LIN {X 0,Y 735.918,Z 1197.735,A -85,B 0,C 180,E1 27996.24,E2 27996.24} C_VEL
LIN {X 0,Y 735.912,Z 1201.928,A -85,B 0,C 180,E1 27994.051,E2 27994.051} C_VEL
LIN {X 0,Y 735.912,Z 1204.213,A -85,B 0,C 180,E1 27992.024,E2 27992.024} C_VEL
LIN {X 0,Y 735.898,Z 1204.939,A -85,B 0,C 180,E1 27989.766,E2 27989.766} C_VEL
LIN {X 0,Y 735.908,Z 1203.976,A -85,B 0,C 180,E1 27987.664,E2 27987.664} C_VEL
LIN {X 0,Y 735.91,Z 1201.303,A -85,B 0,C 180,E1 27985.558,E2 27985.558} C_VEL
LIN {X 0,Y 735.921,Z 1197.152,A -85,B 0,C 180,E1 27983.525,E2 27983.525} C_VEL
LIN {X 0,Y 735.931,Z 1191.15,A -85,B 0,C 180,E1 27981.405,E2 27981.405} C_VEL
LIN {X 0,Y 735.932,Z 1183.317,A -85,B 0,C 180,E1 27979.272,E2 27979.272} C_VEL
LIN {X 0,Y 735.999,Z 1173.523,A -85,B 0,C 180,E1 27977.126,E2 27977.126} C_VEL
LIN {X 0,Y 736.044,Z 1164.524,A -85,B 0,C 180,E1 27975.445,E2 27975.445} C_VEL
LIN {X 0,Y 736.091,Z 1154.647,A -85,B 0,C 180,E1 27973.817,E2 27973.817} C_VEL
LIN {X 0,Y 736.198,Z 1143.668,A -85,B 0,C 180,E1 27972.206,E2 27972.206} C_VEL
LIN {X 0,Y 736.364,Z 1129.285,A -85,B 0,C 180,E1 27970.321,E2 27970.321} C_VEL
LIN {X 0,Y 736.522,Z 1112.613,A -85,B 0,C 180,E1 27968.414,E2 27968.414} C_VEL
LIN {X 0,Y 736.685,Z 1097.971,A -85,B 0,C 180,E1 27966.905,E2 27966.905} C_VEL
LIN {X 0,Y 736.985,Z 1079.519,A -85,B 0,C 180,E1 27965.184,E2 27965.184} C_VEL
LIN {X 0,Y 737.229,Z 1060.157,A -85,B 0,C 180,E1 27963.586,E2 27963.586} C_VEL
LIN {X 0,Y 737.478,Z 1042.502,A -85,B 0,C 180,E1 27962.263,E2 27962.263} C_VEL
LIN {X 0,Y 737.894,Z 1020.414,A -85,B 0,C 180,E1 27960.77,E2 27960.77} C_VEL
LIN {X 0,Y 738.221,Z 997.825,A -85,B 0,C 180,E1 27959.43,E2 27959.43} C_VEL
LIN {X 0,Y 738.518,Z 977.714,A -85,B 0,C 180,E1 27958.361,E2 27958.361} C_VEL
LIN {X 0,Y 738.841,Z 956.603,A -85,B 0,C 180,E1 27957.36,E2 27957.36} C_VEL
LIN {X 0,Y 739.293,Z 929.665,A -85,B 0,C 180,E1 27956.257,E2 27956.257} C_VEL
LIN {X 0,Y 739.568,Z 907.021,A -85,B 0,C 180,E1 27955.471,E2 27955.471} C_VEL
LIN {X 0,Y 739.849,Z 883.645,A -85,B 0,C 180,E1 27954.779,E2 27954.779} C_VEL
LIN {X 0,Y 740.114,Z 856.949,A -85,B 0,C 180,E1 27954.147,E2 27954.147} C_VEL
LIN {X 0,Y 740.323,Z 829.837,A -85,B 0,C 180,E1 27953.669,E2 27953.669} C_VEL
LIN {X 0,Y 740.627,Z 742.145,A -85,B 0,C 180,E1 27952.618,E2 27952.618} C_VEL
LIN {X 0,Y 741.295,Z 519.857,A -85,B 0,C 180,E1 27949.955,E2 27949.955} C_VEL
LIN {X 0,Y 741.706,Z 355.878,A -85,B 0,C 180,E1 27947.919,E2 27947.919} C_VEL
LIN {X 0,Y 740.33,Z 349.95,A -85,B 0,C 180,E1 27947.733,E2 27947.733} C_VEL
LIN {X 0,Y 740.561,Z 322.858,A -85,B 0,C 180,E1 27946.081,E2 27946.081} C_VEL
LIN {X 0,Y 736.124,Z 312.939,A -85,B 0,C 180,E1 27945.097,E2 27945.097} C_VEL
LIN {X 0,Y 736.083,Z 312.459,A -85,B 0,C 180,E1 27944.721,E2 27944.721} C_VEL
LIN {X 0,Y 736.009,Z 312.546,A -85,B 0,C 180,E1 27941.944,E2 27941.944} C_VEL
LIN {X 0,Y 736.01,Z 312.538,A -85,B 0,C 180,E1 27939.58,E2 27939.58} C_VEL
LIN {X 0,Y 736.061,Z 312.541,A -85,B 0,C 180,E1 27936.989,E2 27936.989} C_VEL
LIN {X 0,Y 736.039,Z 312.539,A -85,B 0,C 180,E1 27934.035,E2 27934.035} C_VEL
LIN {X 0,Y 736.022,Z 312.539,A -85,B 0,C 180,E1 27931.536,E2 27931.536} C_VEL
LIN {X 0,Y 736.063,Z 312.544,A -85,B 0,C 180,E1 27928.921,E2 27928.921} C_VEL
LIN {X 0,Y 736.051,Z 312.538,A -85,B 0,C 180,E1 27925.853,E2 27925.853} C_VEL
LIN {X 0,Y 736.033,Z 312.534,A -85,B 0,C 180,E1 27923.286,E2 27923.286} C_VEL
LIN {X 0,Y 736.101,Z 312.542,A -85,B 0,C 180,E1 27920.515,E2 27920.515} C_VEL
LIN {X 0,Y 736.05,Z 312.53,A -85,B 0,C 180,E1 27917.552,E2 27917.552} C_VEL
LIN {X 0,Y 736.058,Z 312.542,A -85,B 0,C 180,E1 27914.877,E2 27914.877} C_VEL
LIN {X 0,Y 736.097,Z 312.528,A -85,B 0,C 180,E1 27911.916,E2 27911.916} C_VEL
LIN {X 0,Y 736.053,Z 312.538,A -85,B 0,C 180,E1 27909.145,E2 27909.145} C_VEL
LIN {X 0,Y 736.094,Z 312.534,A -85,B 0,C 180,E1 27906.317,E2 27906.317} C_VEL
LIN {X 0,Y 736.075,Z 312.534,A -85,B 0,C 180,E1 27903.349,E2 27903.349} C_VEL
LIN {X 0,Y 736.094,Z 312.536,A -85,B 0,C 180,E1 27900.389,E2 27900.389} C_VEL
LIN {X 0,Y 736.092,Z 312.531,A -85,B 0,C 180,E1 27897.353,E2 27897.353} C_VEL
LIN {X 0,Y 736.092,Z 312.536,A -85,B 0,C 180,E1 27894.309,E2 27894.309} C_VEL
LIN {X 0,Y 736.096,Z 312.53,A -85,B 0,C 180,E1 27891.249,E2 27891.249} C_VEL
LIN {X 0,Y 736.093,Z 312.53,A -85,B 0,C 180,E1 27889.116,E2 27889.116} C_VEL
LIN {X 0,Y 735.07,Z 312.665,A -85,B 0,C 180,E1 27888.516,E2 27888.516} C_VEL
LIN {X 0,Y 728.657,Z 313.451,A -85,B 0,C 180,E1 27886.837,E2 27886.837} C_VEL
LIN {X 0,Y 728.145,Z 313.52,A -85,B 0,C 180,E1 27886.401,E2 27886.401} C_VEL
LIN {X 0,Y 728.13,Z 313.524,A -85,B 0,C 180,E1 27883.567,E2 27883.567} C_VEL
LIN {X 0,Y 728.146,Z 313.517,A -85,B 0,C 180,E1 27880.674,E2 27880.674} C_VEL
LIN {X 0,Y 728.133,Z 313.526,A -85,B 0,C 180,E1 27877.75,E2 27877.75} C_VEL
LIN {X 0,Y 728.157,Z 313.518,A -85,B 0,C 180,E1 27874.806,E2 27874.806} C_VEL
LIN {X 0,Y 728.139,Z 313.522,A -85,B 0,C 180,E1 27871.811,E2 27871.811} C_VEL
LIN {X 0,Y 728.131,Z 313.525,A -85,B 0,C 180,E1 27868.913,E2 27868.913} C_VEL
LIN {X 0,Y 728.15,Z 313.526,A -85,B 0,C 180,E1 27865.831,E2 27865.831} C_VEL
LIN {X 0,Y 728.108,Z 313.521,A -85,B 0,C 180,E1 27863.023,E2 27863.023} C_VEL
LIN {X 0,Y 728.159,Z 313.531,A -85,B 0,C 180,E1 27860.139,E2 27860.139} C_VEL
LIN {X 0,Y 728.104,Z 313.534,A -85,B 0,C 180,E1 27857.281,E2 27857.281} C_VEL
LIN {X 0,Y 728.11,Z 313.537,A -85,B 0,C 180,E1 27854.655,E2 27854.655} C_VEL
LIN {X 0,Y 728.206,Z 313.843,A -85,B 0,C 180,E1 27853.987,E2 27853.987} C_VEL
LIN {X 0,Y 733.658,Z 326.305,A -85,B 0,C 180,E1 27852.727,E2 27852.727} C_VEL
LIN {X 0,Y 733.005,Z 366.435,A -85,B 0,C 180,E1 27850.182,E2 27850.182} C_VEL
LIN {X 0,Y 732.691,Z 396.674,A -85,B 0,C 180,E1 27848.329,E2 27848.329} C_VEL
LIN {X 0,Y 734.354,Z 404.868,A -85,B 0,C 180,E1 27848.118,E2 27848.118} C_VEL
LIN {X 0,Y 733.48,Z 650.838,A -85,B 0,C 180,E1 27845.227,E2 27845.227} C_VEL
LIN {X 0,Y 732.832,Z 829.718,A -85,B 0,C 180,E1 27843.161,E2 27843.161} C_VEL
LIN {X 0,Y 732.642,Z 853.04,A -85,B 0,C 180,E1 27842.782,E2 27842.782} C_VEL
LIN {X 0,Y 732.276,Z 879.242,A -85,B 0,C 180,E1 27842.196,E2 27842.196} C_VEL
LIN {X 0,Y 731.992,Z 900.709,A -85,B 0,C 180,E1 27841.591,E2 27841.591} C_VEL
LIN {X 0,Y 731.677,Z 923.398,A -85,B 0,C 180,E1 27840.828,E2 27840.828} C_VEL
LIN {X 0,Y 731.181,Z 948.746,A -85,B 0,C 180,E1 27839.807,E2 27839.807} C_VEL
LIN {X 0,Y 730.811,Z 969.465,A -85,B 0,C 180,E1 27838.835,E2 27838.835} C_VEL
LIN {X 0,Y 730.408,Z 992.417,A -85,B 0,C 180,E1 27837.606,E2 27837.606} C_VEL
LIN {X 0,Y 729.958,Z 1012.888,A -85,B 0,C 180,E1 27836.347,E2 27836.347} C_VEL
LIN {X 0,Y 729.623,Z 1031.699,A -85,B 0,C 180,E1 27835.053,E2 27835.053} C_VEL
LIN {X 0,Y 729.245,Z 1052.078,A -85,B 0,C 180,E1 27833.467,E2 27833.467} C_VEL
LIN {X 0,Y 728.963,Z 1068.5,A -85,B 0,C 180,E1 27832.033,E2 27832.033} C_VEL
LIN {X 0,Y 728.653,Z 1086.838,A -85,B 0,C 180,E1 27830.231,E2 27830.231} C_VEL
LIN {X 0,Y 728.464,Z 1101.019,A -85,B 0,C 180,E1 27828.652,E2 27828.652} C_VEL
LIN {X 0,Y 728.296,Z 1115.544,A -85,B 0,C 180,E1 27826.839,E2 27826.839} C_VEL
LIN {X 0,Y 728.144,Z 1127.947,A -85,B 0,C 180,E1 27825.042,E2 27825.042} C_VEL
LIN {X 0,Y 728.064,Z 1137.806,A -85,B 0,C 180,E1 27823.421,E2 27823.421} C_VEL
LIN {X 0,Y 728.005,Z 1147.195,A -85,B 0,C 180,E1 27821.648,E2 27821.648} C_VEL
LIN {X 0,Y 727.932,Z 1155.983,A -85,B 0,C 180,E1 27819.647,E2 27819.647} C_VEL
LIN {X 0,Y 727.933,Z 1162.049,A -85,B 0,C 180,E1 27817.957,E2 27817.957} C_VEL
LIN {X 0,Y 727.925,Z 1166.828,A -85,B 0,C 180,E1 27816.309,E2 27816.309} C_VEL
LIN {X 0,Y 727.903,Z 1171.167,A -85,B 0,C 180,E1 27814.333,E2 27814.333} C_VEL
LIN {X 0,Y 727.914,Z 1173.832,A -85,B 0,C 180,E1 27812.283,E2 27812.283} C_VEL
LIN {X 0,Y 727.892,Z 1174.814,A -85,B 0,C 180,E1 27810.63,E2 27810.63} C_VEL
LIN {X 0,Y 727.91,Z 1174.706,A -85,B 0,C 180,E1 27808.898,E2 27808.898} C_VEL
LIN {X 0,Y 727.905,Z 1172.917,A -85,B 0,C 180,E1 27806.772,E2 27806.772} C_VEL
LIN {X 0,Y 727.905,Z 1170.075,A -85,B 0,C 180,E1 27805.036,E2 27805.036} C_VEL
LIN {X 0,Y 727.912,Z 1166.237,A -85,B 0,C 180,E1 27803.374,E2 27803.374} C_VEL
LIN {X 0,Y 727.931,Z 1161.006,A -85,B 0,C 180,E1 27801.628,E2 27801.628} C_VEL
LIN {X 0,Y 727.963,Z 1152.715,A -85,B 0,C 180,E1 27799.474,E2 27799.474} C_VEL
LIN {X 0,Y 728.008,Z 1144.792,A -85,B 0,C 180,E1 27797.789,E2 27797.789} C_VEL
LIN {X 0,Y 728.062,Z 1135.921,A -85,B 0,C 180,E1 27796.161,E2 27796.161} C_VEL
LIN {X 0,Y 728.197,Z 1123.732,A -85,B 0,C 180,E1 27794.225,E2 27794.225} C_VEL
LIN {X 0,Y 728.327,Z 1111.132,A -85,B 0,C 180,E1 27792.503,E2 27792.503} C_VEL
LIN {X 0,Y 728.488,Z 1098.245,A -85,B 0,C 180,E1 27790.934,E2 27790.934} C_VEL
LIN {X 0,Y 728.768,Z 1081.226,A -85,B 0,C 180,E1 27789.101,E2 27789.101} C_VEL
LIN {X 0,Y 728.99,Z 1065.335,A -85,B 0,C 180,E1 27787.589,E2 27787.589} C_VEL
LIN {X 0,Y 729.358,Z 1046.931,A -85,B 0,C 180,E1 27786.017,E2 27786.017} C_VEL
LIN {X 0,Y 729.679,Z 1027.552,A -85,B 0,C 180,E1 27784.561,E2 27784.561} C_VEL
LIN {X 0,Y 730.105,Z 1007.614,A -85,B 0,C 180,E1 27783.22,E2 27783.22} C_VEL
LIN {X 0,Y 730.5,Z 985.362,A -85,B 0,C 180,E1 27781.911,E2 27781.911} C_VEL
LIN {X 0,Y 730.883,Z 965.033,A -85,B 0,C 180,E1 27780.855,E2 27780.855} C_VEL
LIN {X 0,Y 731.384,Z 940.503,A -85,B 0,C 180,E1 27779.75,E2 27779.75} C_VEL
LIN {X 0,Y 731.714,Z 918.291,A -85,B 0,C 180,E1 27778.9,E2 27778.9} C_VEL
LIN {X 0,Y 732.031,Z 896.995,A -85,B 0,C 180,E1 27778.204,E2 27778.204} C_VEL
LIN {X 0,Y 732.443,Z 870.527,A -85,B 0,C 180,E1 27777.5,E2 27777.5} C_VEL
LIN {X 0,Y 732.673,Z 847.388,A -85,B 0,C 180,E1 27777.027,E2 27777.027} C_VEL
LIN {X 0,Y 732.843,Z 826.715,A -85,B 0,C 180,E1 27776.708,E2 27776.708} C_VEL
LIN {X 0,Y 733.746,Z 574.835,A -85,B 0,C 180,E1 27773.8,E2 27773.8} C_VEL
LIN {X 0,Y 734.278,Z 403.614,A -85,B 0,C 180,E1 27771.772,E2 27771.772} C_VEL
LIN {X 0,Y 732.662,Z 396.393,A -85,B 0,C 180,E1 27771.569,E2 27771.569} C_VEL
LIN {X 0,Y 733.269,Z 351.692,A -85,B 0,C 180,E1 27768.806,E2 27768.806} C_VEL
LIN {X 0,Y 733.577,Z 326.119,A -85,B 0,C 180,E1 27767.165,E2 27767.165} C_VEL
LIN {X 0,Y 728.22,Z 313.914,A -85,B 0,C 180,E1 27765.934,E2 27765.934} C_VEL
LIN {X 0,Y 728.105,Z 313.538,A -85,B 0,C 180,E1 27765.346,E2 27765.346} C_VEL
LIN {X 0,Y 728.091,Z 313.533,A -85,B 0,C 180,E1 27762.827,E2 27762.827} C_VEL
LIN {X 0,Y 728.157,Z 313.523,A -85,B 0,C 180,E1 27760.093,E2 27760.093} C_VEL
LIN {X 0,Y 728.116,Z 313.52,A -85,B 0,C 180,E1 27757.174,E2 27757.174} C_VEL
LIN {X 0,Y 728.108,Z 313.532,A -85,B 0,C 180,E1 27754.518,E2 27754.518} C_VEL
LIN {X 0,Y 728.155,Z 313.528,A -85,B 0,C 180,E1 27751.639,E2 27751.639} C_VEL
LIN {X 0,Y 728.114,Z 313.517,A -85,B 0,C 180,E1 27748.817,E2 27748.817} C_VEL
LIN {X 0,Y 728.153,Z 313.534,A -85,B 0,C 180,E1 27745.979,E2 27745.979} C_VEL
LIN {X 0,Y 728.141,Z 313.518,A -85,B 0,C 180,E1 27742.954,E2 27742.954} C_VEL
LIN {X 0,Y 728.146,Z 313.532,A -85,B 0,C 180,E1 27739.994,E2 27739.994} C_VEL
LIN {X 0,Y 728.155,Z 313.519,A -85,B 0,C 180,E1 27736.925,E2 27736.925} C_VEL
LIN {X 0,Y 728.153,Z 313.528,A -85,B 0,C 180,E1 27733.874,E2 27733.874} C_VEL
LIN {X 0,Y 728.156,Z 313.518,A -85,B 0,C 180,E1 27730.763,E2 27730.763} C_VEL
LIN {X 0,Y 728.155,Z 313.525,A -85,B 0,C 180,E1 27727.734,E2 27727.734} C_VEL
LIN {X 0,Y 728.158,Z 313.518,A -85,B 0,C 180,E1 27724.647,E2 27724.647} C_VEL
LIN {X 0,Y 728.153,Z 313.524,A -85,B 0,C 180,E1 27721.574,E2 27721.574} C_VEL
LIN {X 0,Y 728.149,Z 313.518,A -85,B 0,C 180,E1 27718.584,E2 27718.584} C_VEL
LIN {X 0,Y 728.153,Z 313.526,A -85,B 0,C 180,E1 27715.5,E2 27715.5} C_VEL
LIN {X 0,Y 728.132,Z 313.52,A -85,B 0,C 180,E1 27712.583,E2 27712.583} C_VEL
LIN {X 0,Y 728.158,Z 313.529,A -85,B 0,C 180,E1 27709.557,E2 27709.557} C_VEL
LIN {X 0,Y 728.112,Z 313.524,A -85,B 0,C 180,E1 27706.742,E2 27706.742} C_VEL
LIN {X 0,Y 728.158,Z 313.525,A -85,B 0,C 180,E1 27703.896,E2 27703.896} C_VEL
LIN {X 0,Y 728.115,Z 313.529,A -85,B 0,C 180,E1 27701.006,E2 27701.006} C_VEL
LIN {X 0,Y 728.111,Z 313.525,A -85,B 0,C 180,E1 27698.321,E2 27698.321} C_VEL
LIN {X 0,Y 728.155,Z 313.528,A -85,B 0,C 180,E1 27695.326,E2 27695.326} C_VEL
LIN {X 0,Y 728.091,Z 313.524,A -85,B 0,C 180,E1 27692.609,E2 27692.609} C_VEL
LIN {X 0,Y 728.113,Z 313.527,A -85,B 0,C 180,E1 27690.009,E2 27690.009} C_VEL
LIN {X 0,Y 728.108,Z 313.531,A -85,B 0,C 180,E1 27686.896,E2 27686.896} C_VEL
LIN {X 0,Y 728.078,Z 313.529,A -85,B 0,C 180,E1 27684.388,E2 27684.388} C_VEL
LIN {X 0,Y 728.095,Z 313.532,A -85,B 0,C 180,E1 27681.895,E2 27681.895} C_VEL
LIN {X 0,Y 728.103,Z 313.538,A -85,B 0,C 180,E1 27678.811,E2 27678.811} C_VEL
LIN {X 0,Y 728.058,Z 313.479,A -85,B 0,C 180,E1 27676.306,E2 27676.306} C_VEL
LIN {X 0,Y 728.149,Z 313.739,A -85,B 0,C 180,E1 27675.498,E2 27675.498} C_VEL
LIN {X 0,Y 729.852,Z 317.558,A -85,B 0,C 180,E1 27675.076,E2 27675.076} C_VEL
LIN {X 0,Y 734.198,Z 327.033,A -85,B 0,C 180,E1 27674.134,E2 27674.134} C_VEL
LIN {X 0,Y 733.988,Z 350.722,A -85,B 0,C 180,E1 27672.697,E2 27672.697} C_VEL
LIN {X 0,Y 735.844,Z 359.271,A -85,B 0,C 180,E1 27672.451,E2 27672.451} C_VEL
LIN {X 0,Y 734.941,Z 571.806,A -85,B 0,C 180,E1 27669.812,E2 27669.812} C_VEL
LIN {X 0,Y 734.051,Z 797.02,A -85,B 0,C 180,E1 27667.112,E2 27667.112} C_VEL
LIN {X 0,Y 733.834,Z 834.513,A -85,B 0,C 180,E1 27666.633,E2 27666.633} C_VEL
LIN {X 0,Y 733.514,Z 861.516,A -85,B 0,C 180,E1 27666.125,E2 27666.125} C_VEL
LIN {X 0,Y 733.167,Z 887.347,A -85,B 0,C 180,E1 27665.488,E2 27665.488} C_VEL
LIN {X 0,Y 732.728,Z 915.129,A -85,B 0,C 180,E1 27664.627,E2 27664.627} C_VEL
LIN {X 0,Y 732.218,Z 939.479,A -85,B 0,C 180,E1 27663.717,E2 27663.717} C_VEL
LIN {X 0,Y 731.801,Z 960.588,A -85,B 0,C 180,E1 27662.807,E2 27662.807} C_VEL
LIN {X 0,Y 731.387,Z 982.087,A -85,B 0,C 180,E1 27661.758,E2 27661.758} C_VEL
LIN {X 0,Y 730.853,Z 1007.155,A -85,B 0,C 180,E1 27660.365,E2 27660.365} C_VEL
LIN {X 0,Y 730.377,Z 1027.567,A -85,B 0,C 180,E1 27659.077,E2 27659.077} C_VEL
LIN {X 0,Y 729.985,Z 1046.466,A -85,B 0,C 180,E1 27657.756,E2 27657.756} C_VEL
LIN {X 0,Y 729.575,Z 1068.232,A -85,B 0,C 180,E1 27656.055,E2 27656.055} C_VEL
LIN {X 0,Y 729.194,Z 1085.448,A -85,B 0,C 180,E1 27654.549,E2 27654.549} C_VEL
LIN {X 0,Y 728.946,Z 1101.391,A -85,B 0,C 180,E1 27653.012,E2 27653.012} C_VEL
LIN {X 0,Y 728.633,Z 1120.122,A -85,B 0,C 180,E1 27650.987,E2 27650.987} C_VEL
LIN {X 0,Y 728.422,Z 1133.803,A -85,B 0,C 180,E1 27649.318,E2 27649.318} C_VEL
LIN {X 0,Y 728.29,Z 1145.418,A -85,B 0,C 180,E1 27647.745,E2 27647.745} C_VEL
LIN {X 0,Y 728.151,Z 1156.938,A -85,B 0,C 180,E1 27646.005,E2 27646.005} C_VEL
LIN {X 0,Y 728.047,Z 1169.421,A -85,B 0,C 180,E1 27643.825,E2 27643.825} C_VEL
LIN {X 0,Y 727.973,Z 1178.073,A -85,B 0,C 180,E1 27642.05,E2 27642.05} C_VEL
LIN {X 0,Y 727.953,Z 1185.837,A -85,B 0,C 180,E1 27640.206,E2 27640.206} C_VEL
LIN {X 0,Y 727.927,Z 1193.111,A -85,B 0,C 180,E1 27638.054,E2 27638.054} C_VEL
LIN {X 0,Y 727.914,Z 1198.422,A -85,B 0,C 180,E1 27635.992,E2 27635.992} C_VEL
LIN {X 0,Y 727.907,Z 1202.278,A -85,B 0,C 180,E1 27633.859,E2 27633.859} C_VEL
LIN {X 0,Y 727.908,Z 1204.493,A -85,B 0,C 180,E1 27631.653,E2 27631.653} C_VEL
LIN {X 0,Y 727.89,Z 1204.872,A -85,B 0,C 180,E1 27629.528,E2 27629.528} C_VEL
LIN {X 0,Y 727.906,Z 1203.905,A -85,B 0,C 180,E1 27627.559,E2 27627.559} C_VEL
LIN {X 0,Y 727.908,Z 1201.178,A -85,B 0,C 180,E1 27625.43,E2 27625.43} C_VEL
LIN {X 0,Y 727.917,Z 1196.956,A -85,B 0,C 180,E1 27623.374,E2 27623.374} C_VEL
LIN {X 0,Y 727.936,Z 1191.147,A -85,B 0,C 180,E1 27621.31,E2 27621.31} C_VEL
LIN {X 0,Y 727.945,Z 1183.636,A -85,B 0,C 180,E1 27619.233,E2 27619.233} C_VEL
LIN {X 0,Y 728.027,Z 1173.524,A -85,B 0,C 180,E1 27616.983,E2 27616.983} C_VEL
LIN {X 0,Y 728.084,Z 1164.525,A -85,B 0,C 180,E1 27615.282,E2 27615.282} C_VEL
LIN {X 0,Y 728.17,Z 1154.738,A -85,B 0,C 180,E1 27613.651,E2 27613.651} C_VEL
LIN {X 0,Y 728.298,Z 1144.116,A -85,B 0,C 180,E1 27612.07,E2 27612.07} C_VEL
LIN {X 0,Y 728.489,Z 1130.976,A -85,B 0,C 180,E1 27610.318,E2 27610.318} C_VEL
LIN {X 0,Y 728.741,Z 1113.472,A -85,B 0,C 180,E1 27608.264,E2 27608.264} C_VEL
LIN {X 0,Y 728.955,Z 1098.827,A -85,B 0,C 180,E1 27606.732,E2 27606.732} C_VEL
LIN {X 0,Y 729.277,Z 1082.529,A -85,B 0,C 180,E1 27605.183,E2 27605.183} C_VEL
LIN {X 0,Y 729.687,Z 1061.264,A -85,B 0,C 180,E1 27603.379,E2 27603.379} C_VEL
LIN {X 0,Y 730.037,Z 1043.446,A -85,B 0,C 180,E1 27602.025,E2 27602.025} C_VEL
LIN {X 0,Y 730.496,Z 1023.585,A -85,B 0,C 180,E1 27600.658,E2 27600.658} C_VEL
LIN {X 0,Y 731.012,Z 999.734,A -85,B 0,C 180,E1 27599.204,E2 27599.204} C_VEL
LIN {X 0,Y 731.426,Z 978.518,A -85,B 0,C 180,E1 27598.059,E2 27598.059} C_VEL
LIN {X 0,Y 731.863,Z 957.7,A -85,B 0,C 180,E1 27597.061,E2 27597.061} C_VEL
LIN {X 0,Y 732.437,Z 932.71,A -85,B 0,C 180,E1 27596.012,E2 27596.012} C_VEL
LIN {X 0,Y 732.846,Z 907.011,A -85,B 0,C 180,E1 27595.109,E2 27595.109} C_VEL
LIN {X 0,Y 733.217,Z 883.845,A -85,B 0,C 180,E1 27594.418,E2 27594.418} C_VEL
LIN {X 0,Y 733.571,Z 857.49,A -85,B 0,C 180,E1 27593.789,E2 27593.789} C_VEL
LIN {X 0,Y 733.853,Z 830.233,A -85,B 0,C 180,E1 27593.303,E2 27593.303} C_VEL
LIN {X 0,Y 734.218,Z 752.07,A -85,B 0,C 180,E1 27592.356,E2 27592.356} C_VEL
LIN {X 0,Y 735.122,Z 528.891,A -85,B 0,C 180,E1 27589.663,E2 27589.663} C_VEL
LIN {X 0,Y 735.759,Z 358.013,A -85,B 0,C 180,E1 27587.527,E2 27587.527} C_VEL
LIN {X 0,Y 733.866,Z 349.652,A -85,B 0,C 180,E1 27587.256,E2 27587.256} C_VEL
LIN {X 0,Y 734.024,Z 326.577,A -85,B 0,C 180,E1 27585.824,E2 27585.824} C_VEL
LIN {X 0,Y 728.179,Z 313.889,A -85,B 0,C 180,E1 27584.529,E2 27584.529} C_VEL
LIN {X 0,Y 728.063,Z 313.458,A -85,B 0,C 180,E1 27584.089,E2 27584.089} C_VEL
LIN {X 0,Y 728.067,Z 313.537,A -85,B 0,C 180,E1 27581.66,E2 27581.66} C_VEL
LIN {X 0,Y 728.114,Z 313.527,A -85,B 0,C 180,E1 27579.074,E2 27579.074} C_VEL
LIN {X 0,Y 728.1,Z 313.527,A -85,B 0,C 180,E1 27576.096,E2 27576.096} C_VEL
LIN {X 0,Y 728.08,Z 313.53,A -85,B 0,C 180,E1 27573.604,E2 27573.604} C_VEL
LIN {X 0,Y 728.117,Z 313.53,A -85,B 0,C 180,E1 27570.996,E2 27570.996} C_VEL
LIN {X 0,Y 728.111,Z 313.521,A -85,B 0,C 180,E1 27567.923,E2 27567.923} C_VEL
LIN {X 0,Y 728.093,Z 313.53,A -85,B 0,C 180,E1 27565.362,E2 27565.362} C_VEL
LIN {X 0,Y 728.153,Z 313.523,A -85,B 0,C 180,E1 27562.612,E2 27562.612} C_VEL
LIN {X 0,Y 728.115,Z 313.525,A -85,B 0,C 180,E1 27559.661,E2 27559.661} C_VEL
LIN {X 0,Y 728.115,Z 313.523,A -85,B 0,C 180,E1 27556.926,E2 27556.926} C_VEL
LIN {X 0,Y 728.158,Z 313.52,A -85,B 0,C 180,E1 27553.986,E2 27553.986} C_VEL
LIN {X 0,Y 728.111,Z 313.52,A -85,B 0,C 180,E1 27551.165,E2 27551.165} C_VEL
LIN {X 0,Y 728.159,Z 313.529,A -85,B 0,C 180,E1 27548.37,E2 27548.37} C_VEL
LIN {X 0,Y 728.131,Z 313.516,A -85,B 0,C 180,E1 27545.358,E2 27545.358} C_VEL
LIN {X 0,Y 728.151,Z 313.533,A -85,B 0,C 180,E1 27542.44,E2 27542.44} C_VEL
LIN {X 0,Y 728.15,Z 313.512,A -85,B 0,C 180,E1 27539.371,E2 27539.371} C_VEL
LIN {X 0,Y 728.151,Z 313.532,A -85,B 0,C 180,E1 27536.378,E2 27536.378} C_VEL
LIN {X 0,Y 728.156,Z 313.51,A -85,B 0,C 180,E1 27533.297,E2 27533.297} C_VEL
LIN {X 0,Y 728.157,Z 313.532,A -85,B 0,C 180,E1 27530.196,E2 27530.196} C_VEL
LIN {X 0,Y 728.155,Z 313.51,A -85,B 0,C 180,E1 27527.147,E2 27527.147} C_VEL
LIN {X 0,Y 728.145,Z 313.52,A -85,B 0,C 180,E1 27526.401,E2 27526.401} C_VEL
LIN {X 0,Y 727.175,Z 313.651,A -85,B 0,C 180,E1 27525.795,E2 27525.795} C_VEL
LIN {X 0,Y 720.732,Z 314.456,A -85,B 0,C 180,E1 27524.097,E2 27524.097} C_VEL
LIN {X 0,Y 720.192,Z 314.514,A -85,B 0,C 180,E1 27523.656,E2 27523.656} C_VEL
LIN {X 0,Y 720.209,Z 314.503,A -85,B 0,C 180,E1 27520.744,E2 27520.744} C_VEL
LIN {X 0,Y 720.198,Z 314.515,A -85,B 0,C 180,E1 27517.813,E2 27517.813} C_VEL
LIN {X 0,Y 720.215,Z 314.507,A -85,B 0,C 180,E1 27514.847,E2 27514.847} C_VEL
LIN {X 0,Y 720.203,Z 314.509,A -85,B 0,C 180,E1 27511.833,E2 27511.833} C_VEL
LIN {X 0,Y 720.191,Z 314.515,A -85,B 0,C 180,E1 27508.938,E2 27508.938} C_VEL
LIN {X 0,Y 720.216,Z 314.511,A -85,B 0,C 180,E1 27505.883,E2 27505.883} C_VEL
LIN {X 0,Y 720.169,Z 314.509,A -85,B 0,C 180,E1 27503.045,E2 27503.045} C_VEL
LIN {X 0,Y 720.22,Z 314.52,A -85,B 0,C 180,E1 27500.15,E2 27500.15} C_VEL
LIN {X 0,Y 720.164,Z 314.523,A -85,B 0,C 180,E1 27497.262,E2 27497.262} C_VEL
LIN {X 0,Y 720.184,Z 314.597,A -85,B 0,C 180,E1 27494.609,E2 27494.609} C_VEL
LIN {X 0,Y 720.441,Z 315.737,A -85,B 0,C 180,E1 27494.433,E2 27494.433} C_VEL
LIN {X 0,Y 727.094,Z 330.153,A -85,B 0,C 180,E1 27492.95,E2 27492.95} C_VEL
LIN {X 0,Y 726.333,Z 368.869,A -85,B 0,C 180,E1 27490.472,E2 27490.472} C_VEL
LIN {X 0,Y 725.991,Z 396.957,A -85,B 0,C 180,E1 27488.742,E2 27488.742} C_VEL
LIN {X 0,Y 728.047,Z 406.7,A -85,B 0,C 180,E1 27488.487,E2 27488.487} C_VEL
LIN {X 0,Y 726.928,Z 654.042,A -85,B 0,C 180,E1 27485.555,E2 27485.555} C_VEL
LIN {X 0,Y 726.124,Z 829.869,A -85,B 0,C 180,E1 27483.506,E2 27483.506} C_VEL
LIN {X 0,Y 725.879,Z 854.455,A -85,B 0,C 180,E1 27483.102,E2 27483.102} C_VEL
LIN {X 0,Y 725.422,Z 880.021,A -85,B 0,C 180,E1 27482.517,E2 27482.517} C_VEL
LIN {X 0,Y 725.065,Z 901.464,A -85,B 0,C 180,E1 27481.905,E2 27481.905} C_VEL
LIN {X 0,Y 724.641,Z 925.926,A -85,B 0,C 180,E1 27481.068,E2 27481.068} C_VEL
LIN {X 0,Y 724.044,Z 949.756,A -85,B 0,C 180,E1 27480.085,E2 27480.085} C_VEL
LIN {X 0,Y 723.572,Z 970.37,A -85,B 0,C 180,E1 27479.105,E2 27479.105} C_VEL
LIN {X 0,Y 723.01,Z 994.628,A -85,B 0,C 180,E1 27477.778,E2 27477.778} C_VEL
LIN {X 0,Y 722.495,Z 1014.222,A -85,B 0,C 180,E1 27476.552,E2 27476.552} C_VEL
LIN {X 0,Y 722.031,Z 1035.1,A -85,B 0,C 180,E1 27475.084,E2 27475.084} C_VEL
LIN {X 0,Y 721.565,Z 1054.043,A -85,B 0,C 180,E1 27473.564,E2 27473.564} C_VEL
LIN {X 0,Y 721.199,Z 1072.131,A -85,B 0,C 180,E1 27471.948,E2 27471.948} C_VEL
LIN {X 0,Y 720.832,Z 1088.401,A -85,B 0,C 180,E1 27470.291,E2 27470.291} C_VEL
LIN {X 0,Y 720.6,Z 1102.442,A -85,B 0,C 180,E1 27468.695,E2 27468.695} C_VEL
LIN {X 0,Y 720.363,Z 1117.879,A -85,B 0,C 180,E1 27466.698,E2 27466.698} C_VEL
LIN {X 0,Y 720.199,Z 1128.994,A -85,B 0,C 180,E1 27465.048,E2 27465.048} C_VEL
LIN {X 0,Y 720.1,Z 1138.738,A -85,B 0,C 180,E1 27463.408,E2 27463.408} C_VEL
LIN {X 0,Y 720.014,Z 1149.201,A -85,B 0,C 180,E1 27461.353,E2 27461.353} C_VEL
LIN {X 0,Y 719.947,Z 1156.9,A -85,B 0,C 180,E1 27459.513,E2 27459.513} C_VEL
LIN {X 0,Y 719.937,Z 1162.504,A -85,B 0,C 180,E1 27457.903,E2 27457.903} C_VEL
LIN {X 0,Y 719.922,Z 1167.45,A -85,B 0,C 180,E1 27456.139,E2 27456.139} C_VEL
LIN {X 0,Y 719.916,Z 1171.774,A -85,B 0,C 180,E1 27453.982,E2 27453.982} C_VEL
LIN {X 0,Y 719.914,Z 1173.9,A -85,B 0,C 180,E1 27452.229,E2 27452.229} C_VEL
LIN {X 0,Y 719.89,Z 1174.859,A -85,B 0,C 180,E1 27450.478,E2 27450.478} C_VEL
LIN {X 0,Y 719.908,Z 1174.579,A -85,B 0,C 180,E1 27448.488,E2 27448.488} C_VEL
LIN {X 0,Y 719.892,Z 1172.578,A -85,B 0,C 180,E1 27446.496,E2 27446.496} C_VEL
LIN {X 0,Y 719.918,Z 1169.662,A -85,B 0,C 180,E1 27444.774,E2 27444.774} C_VEL
LIN {X 0,Y 719.922,Z 1165.203,A -85,B 0,C 180,E1 27442.9,E2 27442.9} C_VEL
LIN {X 0,Y 719.957,Z 1158.461,A -85,B 0,C 180,E1 27440.81,E2 27440.81} C_VEL
LIN {X 0,Y 719.97,Z 1151.645,A -85,B 0,C 180,E1 27439.113,E2 27439.113} C_VEL
LIN {X 0,Y 720.051,Z 1143.921,A -85,B 0,C 180,E1 27437.479,E2 27437.479} C_VEL
LIN {X 0,Y 720.177,Z 1133.194,A -85,B 0,C 180,E1 27435.528,E2 27435.528} C_VEL
LIN {X 0,Y 720.3,Z 1120.834,A -85,B 0,C 180,E1 27433.633,E2 27433.633} C_VEL
LIN {X 0,Y 720.478,Z 1109.2,A -85,B 0,C 180,E1 27432.056,E2 27432.056} C_VEL
LIN {X 0,Y 720.771,Z 1093.251,A -85,B 0,C 180,E1 27430.146,E2 27430.146} C_VEL
LIN {X 0,Y 721.047,Z 1077.677,A -85,B 0,C 180,E1 27428.512,E2 27428.512} C_VEL
LIN {X 0,Y 721.474,Z 1059.669,A -85,B 0,C 180,E1 27426.822,E2 27426.822} C_VEL
LIN {X 0,Y 721.868,Z 1040.84,A -85,B 0,C 180,E1 27425.272,E2 27425.272} C_VEL
LIN {X 0,Y 722.384,Z 1020.837,A -85,B 0,C 180,E1 27423.798,E2 27423.798} C_VEL
LIN {X 0,Y 722.836,Z 1000.103,A -85,B 0,C 180,E1 27422.46,E2 27422.46} C_VEL
LIN {X 0,Y 723.343,Z 980.539,A -85,B 0,C 180,E1 27421.337,E2 27421.337} C_VEL
LIN {X 0,Y 723.926,Z 956.696,A -85,B 0,C 180,E1 27420.138,E2 27420.138} C_VEL
LIN {X 0,Y 724.371,Z 934.898,A -85,B 0,C 180,E1 27419.196,E2 27419.196} C_VEL
LIN {X 0,Y 724.844,Z 913.174,A -85,B 0,C 180,E1 27418.387,E2 27418.387} C_VEL
LIN {X 0,Y 725.365,Z 887.118,A -85,B 0,C 180,E1 27417.583,E2 27417.583} C_VEL
LIN {X 0,Y 725.683,Z 864.784,A -85,B 0,C 180,E1 27417.03,E2 27417.03} C_VEL
LIN {X 0,Y 725.955,Z 843.123,A -85,B 0,C 180,E1 27416.606,E2 27416.606} C_VEL
LIN {X 0,Y 726.229,Z 815.299,A -85,B 0,C 180,E1 27416.215,E2 27416.215} C_VEL
LIN {X 0,Y 727.281,Z 573.749,A -85,B 0,C 180,E1 27413.414,E2 27413.414} C_VEL
LIN {X 0,Y 727.967,Z 405.411,A -85,B 0,C 180,E1 27411.402,E2 27411.402} C_VEL
LIN {X 0,Y 725.906,Z 396.268,A -85,B 0,C 180,E1 27411.141,E2 27411.141} C_VEL
LIN {X 0,Y 726.716,Z 350.874,A -85,B 0,C 180,E1 27408.3,E2 27408.3} C_VEL
LIN {X 0,Y 727.1,Z 330.19,A -85,B 0,C 180,E1 27406.963,E2 27406.963} C_VEL
LIN {X 0,Y 721.261,Z 317.605,A -85,B 0,C 180,E1 27405.671,E2 27405.671} C_VEL
LIN {X 0,Y 720.189,Z 314.7,A -85,B 0,C 180,E1 27405.34,E2 27405.34} C_VEL
LIN {X 0,Y 720.152,Z 314.523,A -85,B 0,C 180,E1 27402.854,E2 27402.854} C_VEL
LIN {X 0,Y 720.216,Z 314.51,A -85,B 0,C 180,E1 27400.097,E2 27400.097} C_VEL
LIN {X 0,Y 720.175,Z 314.508,A -85,B 0,C 180,E1 27397.154,E2 27397.154} C_VEL
LIN {X 0,Y 720.174,Z 314.522,A -85,B 0,C 180,E1 27394.442,E2 27394.442} C_VEL
LIN {X 0,Y 720.222,Z 314.514,A -85,B 0,C 180,E1 27391.467,E2 27391.467} C_VEL
LIN {X 0,Y 720.171,Z 314.506,A -85,B 0,C 180,E1 27388.62,E2 27388.62} C_VEL
LIN {X 0,Y 720.217,Z 314.518,A -85,B 0,C 180,E1 27385.845,E2 27385.845} C_VEL
LIN {X 0,Y 720.191,Z 314.508,A -85,B 0,C 180,E1 27382.8,E2 27382.8} C_VEL
LIN {X 0,Y 720.216,Z 314.515,A -85,B 0,C 180,E1 27379.885,E2 27379.885} C_VEL
LIN {X 0,Y 720.205,Z 314.509,A -85,B 0,C 180,E1 27376.785,E2 27376.785} C_VEL
LIN {X 0,Y 720.217,Z 314.513,A -85,B 0,C 180,E1 27373.815,E2 27373.815} C_VEL
LIN {X 0,Y 720.215,Z 314.507,A -85,B 0,C 180,E1 27370.722,E2 27370.722} C_VEL
LIN {X 0,Y 720.215,Z 314.51,A -85,B 0,C 180,E1 27367.659,E2 27367.659} C_VEL
LIN {X 0,Y 720.219,Z 314.507,A -85,B 0,C 180,E1 27364.59,E2 27364.59} C_VEL
LIN {X 0,Y 720.21,Z 314.51,A -85,B 0,C 180,E1 27361.512,E2 27361.512} C_VEL
LIN {X 0,Y 720.217,Z 314.506,A -85,B 0,C 180,E1 27358.488,E2 27358.488} C_VEL
LIN {X 0,Y 720.202,Z 314.512,A -85,B 0,C 180,E1 27355.381,E2 27355.381} C_VEL
LIN {X 0,Y 720.208,Z 314.506,A -85,B 0,C 180,E1 27352.417,E2 27352.417} C_VEL
LIN {X 0,Y 720.204,Z 314.513,A -85,B 0,C 180,E1 27349.359,E2 27349.359} C_VEL
LIN {X 0,Y 720.181,Z 314.51,A -85,B 0,C 180,E1 27346.511,E2 27346.511} C_VEL
LIN {X 0,Y 720.219,Z 314.516,A -85,B 0,C 180,E1 27343.548,E2 27343.548} C_VEL
LIN {X 0,Y 720.165,Z 314.516,A -85,B 0,C 180,E1 27340.704,E2 27340.704} C_VEL
LIN {X 0,Y 720.221,Z 314.512,A -85,B 0,C 180,E1 27337.899,E2 27337.899} C_VEL
LIN {X 0,Y 720.172,Z 314.522,A -85,B 0,C 180,E1 27334.946,E2 27334.946} C_VEL
LIN {X 0,Y 720.155,Z 314.51,A -85,B 0,C 180,E1 27332.351,E2 27332.351} C_VEL
LIN {X 0,Y 720.224,Z 314.517,A -85,B 0,C 180,E1 27329.553,E2 27329.553} C_VEL
LIN {X 0,Y 720.149,Z 314.52,A -85,B 0,C 180,E1 27326.645,E2 27326.645} C_VEL
LIN {X 0,Y 720.142,Z 314.517,A -85,B 0,C 180,E1 27324.179,E2 27324.179} C_VEL
LIN {X 0,Y 720.224,Z 314.52,A -85,B 0,C 180,E1 27321.337,E2 27321.337} C_VEL
LIN {X 0,Y 720.138,Z 314.527,A -85,B 0,C 180,E1 27318.524,E2 27318.524} C_VEL
LIN {X 0,Y 720.139,Z 314.62,A -85,B 0,C 180,E1 27316.144,E2 27316.144} C_VEL
LIN {X 0,Y 720.363,Z 315.642,A -85,B 0,C 180,E1 27315.971,E2 27315.971} C_VEL
LIN {X 0,Y 726.297,Z 328.014,A -85,B 0,C 180,E1 27314.678,E2 27314.678} C_VEL
LIN {X 0,Y 727.794,Z 331.004,A -85,B 0,C 180,E1 27314.37,E2 27314.37} C_VEL
LIN {X 0,Y 727.557,Z 350.65,A -85,B 0,C 180,E1 27313.168,E2 27313.168} C_VEL
LIN {X 0,Y 729.916,Z 361.282,A -85,B 0,C 180,E1 27312.851,E2 27312.851} C_VEL
LIN {X 0,Y 728.775,Z 573.944,A -85,B 0,C 180,E1 27310.191,E2 27310.191} C_VEL
LIN {X 0,Y 727.652,Z 799.31,A -85,B 0,C 180,E1 27307.467,E2 27307.467} C_VEL
LIN {X 0,Y 727.385,Z 835.279,A -85,B 0,C 180,E1 27306.999,E2 27306.999} C_VEL
LIN {X 0,Y 726.978,Z 862.571,A -85,B 0,C 180,E1 27306.478,E2 27306.478} C_VEL
LIN {X 0,Y 726.543,Z 888.174,A -85,B 0,C 180,E1 27305.837,E2 27305.837} C_VEL
LIN {X 0,Y 725.974,Z 916.194,A -85,B 0,C 180,E1 27304.956,E2 27304.956} C_VEL
LIN {X 0,Y 725.376,Z 939.91,A -85,B 0,C 180,E1 27304.06,E2 27304.06} C_VEL
LIN {X 0,Y 724.836,Z 961.083,A -85,B 0,C 180,E1 27303.139,E2 27303.139} C_VEL
LIN {X 0,Y 724.298,Z 983.241,A -85,B 0,C 180,E1 27302.045,E2 27302.045} C_VEL
LIN {X 0,Y 723.607,Z 1008.617,A -85,B 0,C 180,E1 27300.61,E2 27300.61} C_VEL
LIN {X 0,Y 723.048,Z 1028.231,A -85,B 0,C 180,E1 27299.355,E2 27299.355} C_VEL
LIN {X 0,Y 722.54,Z 1047.296,A -85,B 0,C 180,E1 27298.005,E2 27298.005} C_VEL
LIN {X 0,Y 721.988,Z 1069.755,A -85,B 0,C 180,E1 27296.217,E2 27296.217} C_VEL
LIN {X 0,Y 721.544,Z 1086.381,A -85,B 0,C 180,E1 27294.739,E2 27294.739} C_VEL
LIN {X 0,Y 721.207,Z 1103.094,A -85,B 0,C 180,E1 27293.101,E2 27293.101} C_VEL
LIN {X 0,Y 720.82,Z 1120.834,A -85,B 0,C 180,E1 27291.14,E2 27291.14} C_VEL
LIN {X 0,Y 720.583,Z 1133.805,A -85,B 0,C 180,E1 27289.536,E2 27289.536} C_VEL
LIN {X 0,Y 720.389,Z 1146.002,A -85,B 0,C 180,E1 27287.863,E2 27287.863} C_VEL
LIN {X 0,Y 720.214,Z 1158.902,A -85,B 0,C 180,E1 27285.872,E2 27285.872} C_VEL
LIN {X 0,Y 720.078,Z 1170.243,A -85,B 0,C 180,E1 27283.818,E2 27283.818} C_VEL
LIN {X 0,Y 719.995,Z 1178.432,A -85,B 0,C 180,E1 27282.104,E2 27282.104} C_VEL
LIN {X 0,Y 719.965,Z 1186.135,A -85,B 0,C 180,E1 27280.239,E2 27280.239} C_VEL
LIN {X 0,Y 719.933,Z 1193.544,A -85,B 0,C 180,E1 27278.001,E2 27278.001} C_VEL
LIN {X 0,Y 719.918,Z 1198.937,A -85,B 0,C 180,E1 27275.819,E2 27275.819} C_VEL
LIN {X 0,Y 719.909,Z 1202.484,A -85,B 0,C 180,E1 27273.743,E2 27273.743} C_VEL
LIN {X 0,Y 719.909,Z 1204.549,A -85,B 0,C 180,E1 27271.592,E2 27271.592} C_VEL
LIN {X 0,Y 719.89,Z 1204.872,A -85,B 0,C 180,E1 27269.522,E2 27269.522} C_VEL
LIN {X 0,Y 719.906,Z 1203.902,A -85,B 0,C 180,E1 27267.532,E2 27267.532} C_VEL
LIN {X 0,Y 719.908,Z 1201.178,A -85,B 0,C 180,E1 27265.379,E2 27265.379} C_VEL
LIN {X 0,Y 719.916,Z 1196.832,A -85,B 0,C 180,E1 27263.249,E2 27263.249} C_VEL
LIN {X 0,Y 719.938,Z 1190.89,A -85,B 0,C 180,E1 27261.132,E2 27261.132} C_VEL
LIN {X 0,Y 719.972,Z 1182.999,A -85,B 0,C 180,E1 27258.951,E2 27258.951} C_VEL
LIN {X 0,Y 720.061,Z 1173.152,A -85,B 0,C 180,E1 27256.762,E2 27256.762} C_VEL
LIN {X 0,Y 720.128,Z 1164.061,A -85,B 0,C 180,E1 27255.033,E2 27255.033} C_VEL
LIN {X 0,Y 720.263,Z 1154.217,A -85,B 0,C 180,E1 27253.383,E2 27253.383} C_VEL
LIN {X 0,Y 720.436,Z 1142.826,A -85,B 0,C 180,E1 27251.682,E2 27251.682} C_VEL
LIN {X 0,Y 720.711,Z 1127.218,A -85,B 0,C 180,E1 27249.621,E2 27249.621} C_VEL
LIN {X 0,Y 720.991,Z 1111.837,A -85,B 0,C 180,E1 27247.839,E2 27247.839} C_VEL
LIN {X 0,Y 721.335,Z 1096.267,A -85,B 0,C 180,E1 27246.211,E2 27246.211} C_VEL
LIN {X 0,Y 721.804,Z 1075.845,A -85,B 0,C 180,E1 27244.305,E2 27244.305} C_VEL
LIN {X 0,Y 722.251,Z 1058.496,A -85,B 0,C 180,E1 27242.861,E2 27242.861} C_VEL
LIN {X 0,Y 722.773,Z 1039.952,A -85,B 0,C 180,E1 27241.458,E2 27241.458} C_VEL
LIN {X 0,Y 723.392,Z 1015.884,A -85,B 0,C 180,E1 27239.839,E2 27239.839} C_VEL
LIN {X 0,Y 723.928,Z 995.422,A -85,B 0,C 180,E1 27238.62,E2 27238.62} C_VEL
LIN {X 0,Y 724.506,Z 974.96,A -85,B 0,C 180,E1 27237.53,E2 27237.53} C_VEL
LIN {X 0,Y 725.208,Z 949.538,A -85,B 0,C 180,E1 27236.34,E2 27236.34} C_VEL
LIN {X 0,Y 725.729,Z 925.114,A -85,B 0,C 180,E1 27235.366,E2 27235.366} C_VEL
LIN {X 0,Y 726.184,Z 904.097,A -85,B 0,C 180,E1 27234.645,E2 27234.645} C_VEL
LIN {X 0,Y 726.663,Z 880.878,A -85,B 0,C 180,E1 27233.965,E2 27233.965} C_VEL
LIN {X 0,Y 727.133,Z 854.027,A -85,B 0,C 180,E1 27233.341,E2 27233.341} C_VEL
LIN {X 0,Y 727.453,Z 827.025,A -85,B 0,C 180,E1 27232.878,E2 27232.878} C_VEL
LIN {X 0,Y 728.67,Z 592.893,A -85,B 0,C 180,E1 27230.042,E2 27230.042} C_VEL
LIN {X 0,Y 729.756,Z 386.877,A -85,B 0,C 180,E1 27227.473,E2 27227.473} C_VEL
LIN {X 0,Y 729.741,Z 359.659,A -85,B 0,C 180,E1 27227.115,E2 27227.115} C_VEL
LIN {X 0,Y 727.454,Z 349.739,A -85,B 0,C 180,E1 27226.792,E2 27226.792} C_VEL
LIN {X 0,Y 727.66,Z 330.784,A -85,B 0,C 180,E1 27225.606,E2 27225.606} C_VEL
LIN {X 0,Y 721.58,Z 318.115,A -85,B 0,C 180,E1 27224.298,E2 27224.298} C_VEL
LIN {X 0,Y 720.159,Z 314.746,A -85,B 0,C 180,E1 27223.913,E2 27223.913} C_VEL
LIN {X 0,Y 720.212,Z 314.489,A -85,B 0,C 180,E1 27222.742,E2 27222.742} C_VEL
LIN {X 0,Y 720.137,Z 314.513,A -85,B 0,C 180,E1 27219.966,E2 27219.966} C_VEL
LIN {X 0,Y 720.135,Z 314.523,A -85,B 0,C 180,E1 27217.551,E2 27217.551} C_VEL
LIN {X 0,Y 720.212,Z 314.521,A -85,B 0,C 180,E1 27214.792,E2 27214.792} C_VEL
LIN {X 0,Y 720.153,Z 314.515,A -85,B 0,C 180,E1 27211.844,E2 27211.844} C_VEL
LIN {X 0,Y 720.152,Z 314.52,A -85,B 0,C 180,E1 27209.316,E2 27209.316} C_VEL
LIN {X 0,Y 720.221,Z 314.519,A -85,B 0,C 180,E1 27206.554,E2 27206.554} C_VEL
LIN {X 0,Y 720.163,Z 314.507,A -85,B 0,C 180,E1 27203.657,E2 27203.657} C_VEL
LIN {X 0,Y 720.174,Z 314.519,A -85,B 0,C 180,E1 27200.99,E2 27200.99} C_VEL
LIN {X 0,Y 720.217,Z 314.503,A -85,B 0,C 180,E1 27198.013,E2 27198.013} C_VEL
LIN {X 0,Y 720.166,Z 314.518,A -85,B 0,C 180,E1 27195.213,E2 27195.213} C_VEL
LIN {X 0,Y 720.219,Z 314.507,A -85,B 0,C 180,E1 27192.427,E2 27192.427} C_VEL
LIN {X 0,Y 720.187,Z 314.513,A -85,B 0,C 180,E1 27189.429,E2 27189.429} C_VEL
LIN {X 0,Y 720.207,Z 314.51,A -85,B 0,C 180,E1 27186.537,E2 27186.537} C_VEL
LIN {X 0,Y 720.205,Z 314.511,A -85,B 0,C 180,E1 27183.423,E2 27183.423} C_VEL
LIN {X 0,Y 720.206,Z 314.511,A -85,B 0,C 180,E1 27180.477,E2 27180.477} C_VEL
LIN {X 0,Y 720.215,Z 314.509,A -85,B 0,C 180,E1 27177.374,E2 27177.374} C_VEL
LIN {X 0,Y 720.213,Z 314.51,A -85,B 0,C 180,E1 27174.343,E2 27174.343} C_VEL
LIN {X 0,Y 720.218,Z 314.508,A -85,B 0,C 180,E1 27171.216,E2 27171.216} C_VEL
LIN {X 0,Y 720.215,Z 314.507,A -85,B 0,C 180,E1 27168.143,E2 27168.143} C_VEL
LIN {X 0,Y 720.218,Z 314.509,A -85,B 0,C 180,E1 27165.074,E2 27165.074} C_VEL
LIN {X 0,Y 720.192,Z 314.514,A -85,B 0,C 180,E1 27163.656,E2 27163.656} C_VEL
LIN {X 0,Y 719.204,Z 314.635,A -85,B 0,C 180,E1 27163.043,E2 27163.043} C_VEL
LIN {X 0,Y 712.81,Z 315.423,A -85,B 0,C 180,E1 27161.326,E2 27161.326} C_VEL
LIN {X 0,Y 712.275,Z 315.489,A -85,B 0,C 180,E1 27160.88,E2 27160.88} C_VEL
LIN {X 0,Y 712.266,Z 315.504,A -85,B 0,C 180,E1 27157.897,E2 27157.897} C_VEL
LIN {X 0,Y 712.273,Z 315.496,A -85,B 0,C 180,E1 27154.883,E2 27154.883} C_VEL
LIN {X 0,Y 712.258,Z 315.495,A -85,B 0,C 180,E1 27151.765,E2 27151.765} C_VEL
LIN {X 0,Y 712.256,Z 315.504,A -85,B 0,C 180,E1 27148.895,E2 27148.895} C_VEL
LIN {X 0,Y 712.264,Z 315.502,A -85,B 0,C 180,E1 27145.776,E2 27145.776} C_VEL
LIN {X 0,Y 712.233,Z 315.496,A -85,B 0,C 180,E1 27142.967,E2 27142.967} C_VEL
LIN {X 0,Y 712.281,Z 315.501,A -85,B 0,C 180,E1 27139.989,E2 27139.989} C_VEL
LIN {X 0,Y 712.224,Z 315.513,A -85,B 0,C 180,E1 27137.196,E2 27137.196} C_VEL
LIN {X 0,Y 712.241,Z 315.675,A -85,B 0,C 180,E1 27135.149,E2 27135.149} C_VEL
LIN {X 0,Y 713.666,Z 319.191,A -85,B 0,C 180,E1 27134.737,E2 27134.737} C_VEL
LIN {X 0,Y 720.578,Z 334.352,A -85,B 0,C 180,E1 27133.151,E2 27133.151} C_VEL
LIN {X 0,Y 719.601,Z 375.037,A -85,B 0,C 180,E1 27130.53,E2 27130.53} C_VEL
LIN {X 0,Y 719.207,Z 396.41,A -85,B 0,C 180,E1 27129.194,E2 27129.194} C_VEL
LIN {X 0,Y 721.769,Z 408.53,A -85,B 0,C 180,E1 27128.862,E2 27128.862} C_VEL
LIN {X 0,Y 720.407,Z 655.747,A -85,B 0,C 180,E1 27125.907,E2 27125.907} C_VEL
LIN {X 0,Y 719.444,Z 829.913,A -85,B 0,C 180,E1 27123.859,E2 27123.859} C_VEL
LIN {X 0,Y 719.141,Z 854.924,A -85,B 0,C 180,E1 27123.444,E2 27123.444} C_VEL
LIN {X 0,Y 718.599,Z 880.42,A -85,B 0,C 180,E1 27122.855,E2 27122.855} C_VEL
LIN {X 0,Y 718.16,Z 902.22,A -85,B 0,C 180,E1 27122.225,E2 27122.225} C_VEL
LIN {X 0,Y 717.593,Z 927.736,A -85,B 0,C 180,E1 27121.333,E2 27121.333} C_VEL
LIN {X 0,Y 716.962,Z 949.773,A -85,B 0,C 180,E1 27120.414,E2 27120.414} C_VEL
LIN {X 0,Y 716.364,Z 970.386,A -85,B 0,C 180,E1 27119.427,E2 27119.427} C_VEL
LIN {X 0,Y 715.695,Z 994.633,A -85,B 0,C 180,E1 27118.087,E2 27118.087} C_VEL
LIN {X 0,Y 715.088,Z 1014.233,A -85,B 0,C 180,E1 27116.849,E2 27116.849} C_VEL
LIN {X 0,Y 714.515,Z 1034.71,A -85,B 0,C 180,E1 27115.399,E2 27115.399} C_VEL
LIN {X 0,Y 713.961,Z 1053.685,A -85,B 0,C 180,E1 27113.862,E2 27113.862} C_VEL
LIN {X 0,Y 713.505,Z 1070.828,A -85,B 0,C 180,E1 27112.32,E2 27112.32} C_VEL
LIN {X 0,Y 713.081,Z 1087.63,A -85,B 0,C 180,E1 27110.607,E2 27110.607} C_VEL
LIN {X 0,Y 712.766,Z 1101.74,A -85,B 0,C 180,E1 27108.993,E2 27108.993} C_VEL
LIN {X 0,Y 712.485,Z 1116.723,A -85,B 0,C 180,E1 27107.056,E2 27107.056} C_VEL
LIN {X 0,Y 712.284,Z 1128.478,A -85,B 0,C 180,E1 27105.302,E2 27105.302} C_VEL
LIN {X 0,Y 712.144,Z 1138.279,A -85,B 0,C 180,E1 27103.644,E2 27103.644} C_VEL
LIN {X 0,Y 712.05,Z 1148.4,A -85,B 0,C 180,E1 27101.666,E2 27101.666} C_VEL
LIN {X 0,Y 711.952,Z 1156.598,A -85,B 0,C 180,E1 27099.703,E2 27099.703} C_VEL
LIN {X 0,Y 711.943,Z 1162.322,A -85,B 0,C 180,E1 27098.051,E2 27098.051} C_VEL
LIN {X 0,Y 711.928,Z 1167.245,A -85,B 0,C 180,E1 27096.289,E2 27096.289} C_VEL
LIN {X 0,Y 711.916,Z 1171.661,A -85,B 0,C 180,E1 27094.108,E2 27094.108} C_VEL
LIN {X 0,Y 711.915,Z 1173.9,A -85,B 0,C 180,E1 27092.254,E2 27092.254} C_VEL
LIN {X 0,Y 711.89,Z 1174.859,A -85,B 0,C 180,E1 27090.483,E2 27090.483} C_VEL
LIN {X 0,Y 711.907,Z 1174.579,A -85,B 0,C 180,E1 27088.471,E2 27088.471} C_VEL
LIN {X 0,Y 711.892,Z 1172.578,A -85,B 0,C 180,E1 27086.457,E2 27086.457} C_VEL
LIN {X 0,Y 711.918,Z 1169.721,A -85,B 0,C 180,E1 27084.745,E2 27084.745} C_VEL
LIN {X 0,Y 711.924,Z 1165.408,A -85,B 0,C 180,E1 27082.901,E2 27082.901} C_VEL
LIN {X 0,Y 711.966,Z 1158.459,A -85,B 0,C 180,E1 27080.706,E2 27080.706} C_VEL
LIN {X 0,Y 711.99,Z 1151.644,A -85,B 0,C 180,E1 27078.99,E2 27078.99} C_VEL
LIN {X 0,Y 712.085,Z 1143.97,A -85,B 0,C 180,E1 27077.347,E2 27077.347} C_VEL
LIN {X 0,Y 712.234,Z 1133.19,A -85,B 0,C 180,E1 27075.363,E2 27075.363} C_VEL
LIN {X 0,Y 712.403,Z 1120.832,A -85,B 0,C 180,E1 27073.446,E2 27073.446} C_VEL
LIN {X 0,Y 712.623,Z 1108.555,A -85,B 0,C 180,E1 27071.767,E2 27071.767} C_VEL
LIN {X 0,Y 712.967,Z 1092.336,A -85,B 0,C 180,E1 27069.819,E2 27069.819} C_VEL
LIN {X 0,Y 713.317,Z 1077.808,A -85,B 0,C 180,E1 27068.281,E2 27068.281} C_VEL
LIN {X 0,Y 713.815,Z 1059.73,A -85,B 0,C 180,E1 27066.565,E2 27066.565} C_VEL
LIN {X 0,Y 714.317,Z 1040.834,A -85,B 0,C 180,E1 27064.993,E2 27064.993} C_VEL
LIN {X 0,Y 714.927,Z 1020.826,A -85,B 0,C 180,E1 27063.504,E2 27063.504} C_VEL
LIN {X 0,Y 715.515,Z 999.74,A -85,B 0,C 180,E1 27062.132,E2 27062.132} C_VEL
LIN {X 0,Y 716.134,Z 979.716,A -85,B 0,C 180,E1 27060.976,E2 27060.976} C_VEL
LIN {X 0,Y 716.818,Z 955.04,A -85,B 0,C 180,E1 27059.735,E2 27059.735} C_VEL
LIN {X 0,Y 717.382,Z 933.771,A -85,B 0,C 180,E1 27058.816,E2 27058.816} C_VEL
LIN {X 0,Y 718.012,Z 910.581,A -85,B 0,C 180,E1 27057.956,E2 27057.956} C_VEL
LIN {X 0,Y 718.55,Z 884.63,A -85,B 0,C 180,E1 27057.169,E2 27057.169} C_VEL
LIN {X 0,Y 718.934,Z 862.826,A -85,B 0,C 180,E1 27056.636,E2 27056.636} C_VEL
LIN {X 0,Y 719.359,Z 838.161,A -85,B 0,C 180,E1 27056.168,E2 27056.168} C_VEL
LIN {X 0,Y 719.633,Z 802.517,A -85,B 0,C 180,E1 27055.713,E2 27055.713} C_VEL
LIN {X 0,Y 720.877,Z 566.492,A -85,B 0,C 180,E1 27052.947,E2 27052.947} C_VEL
LIN {X 0,Y 721.677,Z 407.208,A -85,B 0,C 180,E1 27051.026,E2 27051.026} C_VEL
LIN {X 0,Y 719.207,Z 396.373,A -85,B 0,C 180,E1 27050.715,E2 27050.715} C_VEL
LIN {X 0,Y 720.209,Z 350.053,A -85,B 0,C 180,E1 27047.783,E2 27047.783} C_VEL
LIN {X 0,Y 720.58,Z 334.381,A -85,B 0,C 180,E1 27046.761,E2 27046.761} C_VEL
LIN {X 0,Y 713.859,Z 319.472,A -85,B 0,C 180,E1 27045.208,E2 27045.208} C_VEL
LIN {X 0,Y 712.259,Z 315.834,A -85,B 0,C 180,E1 27044.795,E2 27044.795} C_VEL
LIN {X 0,Y 712.279,Z 315.489,A -85,B 0,C 180,E1 27044.051,E2 27044.051} C_VEL
LIN {X 0,Y 712.227,Z 315.493,A -85,B 0,C 180,E1 27041.18,E2 27041.18} C_VEL
LIN {X 0,Y 712.227,Z 315.513,A -85,B 0,C 180,E1 27038.56,E2 27038.56} C_VEL
LIN {X 0,Y 712.281,Z 315.506,A -85,B 0,C 180,E1 27035.632,E2 27035.632} C_VEL
LIN {X 0,Y 712.227,Z 315.496,A -85,B 0,C 180,E1 27032.763,E2 27032.763} C_VEL
LIN {X 0,Y 712.28,Z 315.501,A -85,B 0,C 180,E1 27029.984,E2 27029.984} C_VEL
LIN {X 0,Y 712.252,Z 315.503,A -85,B 0,C 180,E1 27026.947,E2 27026.947} C_VEL
LIN {X 0,Y 712.266,Z 315.497,A -85,B 0,C 180,E1 27024.023,E2 27024.023} C_VEL
LIN {X 0,Y 712.265,Z 315.501,A -85,B 0,C 180,E1 27020.89,E2 27020.89} C_VEL
LIN {X 0,Y 712.273,Z 315.495,A -85,B 0,C 180,E1 27017.869,E2 27017.869} C_VEL
LIN {X 0,Y 712.275,Z 315.499,A -85,B 0,C 180,E1 27014.803,E2 27014.803} C_VEL
LIN {X 0,Y 712.276,Z 315.495,A -85,B 0,C 180,E1 27011.745,E2 27011.745} C_VEL
LIN {X 0,Y 712.275,Z 315.498,A -85,B 0,C 180,E1 27008.639,E2 27008.639} C_VEL
LIN {X 0,Y 712.271,Z 315.497,A -85,B 0,C 180,E1 27005.559,E2 27005.559} C_VEL
LIN {X 0,Y 712.276,Z 315.499,A -85,B 0,C 180,E1 27002.494,E2 27002.494} C_VEL
LIN {X 0,Y 712.266,Z 315.498,A -85,B 0,C 180,E1 26999.437,E2 26999.437} C_VEL
LIN {X 0,Y 712.276,Z 315.5,A -85,B 0,C 180,E1 26996.451,E2 26996.451} C_VEL
LIN {X 0,Y 712.264,Z 315.497,A -85,B 0,C 180,E1 26993.39,E2 26993.39} C_VEL
LIN {X 0,Y 712.258,Z 315.501,A -85,B 0,C 180,E1 26990.465,E2 26990.465} C_VEL
LIN {X 0,Y 712.264,Z 315.497,A -85,B 0,C 180,E1 26987.327,E2 26987.327} C_VEL
LIN {X 0,Y 712.243,Z 315.504,A -85,B 0,C 180,E1 26984.446,E2 26984.446} C_VEL
LIN {X 0,Y 712.275,Z 315.496,A -85,B 0,C 180,E1 26981.418,E2 26981.418} C_VEL
LIN {X 0,Y 712.224,Z 315.505,A -85,B 0,C 180,E1 26978.591,E2 26978.591} C_VEL
LIN {X 0,Y 712.28,Z 315.492,A -85,B 0,C 180,E1 26975.801,E2 26975.801} C_VEL
LIN {X 0,Y 712.226,Z 315.501,A -85,B 0,C 180,E1 26972.853,E2 26972.853} C_VEL
LIN {X 0,Y 712.215,Z 315.507,A -85,B 0,C 180,E1 26970.292,E2 26970.292} C_VEL
LIN {X 0,Y 712.282,Z 315.494,A -85,B 0,C 180,E1 26967.379,E2 26967.379} C_VEL
LIN {X 0,Y 712.203,Z 315.507,A -85,B 0,C 180,E1 26964.515,E2 26964.515} C_VEL
LIN {X 0,Y 712.206,Z 315.511,A -85,B 0,C 180,E1 26962.053,E2 26962.053} C_VEL
LIN {X 0,Y 712.273,Z 315.5,A -85,B 0,C 180,E1 26959.143,E2 26959.143} C_VEL
LIN {X 0,Y 712.238,Z 315.694,A -85,B 0,C 180,E1 26956.691,E2 26956.691} C_VEL
LIN {X 0,Y 713.558,Z 319.026,A -85,B 0,C 180,E1 26956.304,E2 26956.304} C_VEL
LIN {X 0,Y 718.82,Z 329.838,A -85,B 0,C 180,E1 26955.15,E2 26955.15} C_VEL
LIN {X 0,Y 721.404,Z 335.623,A -85,B 0,C 180,E1 26954.567,E2 26954.567} C_VEL
LIN {X 0,Y 721.093,Z 349.995,A -85,B 0,C 180,E1 26953.672,E2 26953.672} C_VEL
LIN {X 0,Y 724.024,Z 363.321,A -85,B 0,C 180,E1 26953.258,E2 26953.258} C_VEL
LIN {X 0,Y 722.642,Z 575.694,A -85,B 0,C 180,E1 26950.58,E2 26950.58} C_VEL
LIN {X 0,Y 721.287,Z 800.71,A -85,B 0,C 180,E1 26947.838,E2 26947.838} C_VEL
LIN {X 0,Y 720.964,Z 835.688,A -85,B 0,C 180,E1 26947.377,E2 26947.377} C_VEL
LIN {X 0,Y 720.476,Z 862.942,A -85,B 0,C 180,E1 26946.851,E2 26946.851} C_VEL
LIN {X 0,Y 719.964,Z 888.321,A -85,B 0,C 180,E1 26946.211,E2 26946.211} C_VEL
LIN {X 0,Y 719.265,Z 916.703,A -85,B 0,C 180,E1 26945.311,E2 26945.311} C_VEL
LIN {X 0,Y 718.6,Z 939.487,A -85,B 0,C 180,E1 26944.445,E2 26944.445} C_VEL
LIN {X 0,Y 717.941,Z 960.694,A -85,B 0,C 180,E1 26943.518,E2 26943.518} C_VEL
LIN {X 0,Y 717.251,Z 982.984,A -85,B 0,C 180,E1 26942.412,E2 26942.412} C_VEL
LIN {X 0,Y 716.464,Z 1007.885,A -85,B 0,C 180,E1 26940.995,E2 26940.995} C_VEL
LIN {X 0,Y 715.787,Z 1027.571,A -85,B 0,C 180,E1 26939.729,E2 26939.729} C_VEL
LIN {X 0,Y 715.19,Z 1045.813,A -85,B 0,C 180,E1 26938.431,E2 26938.431} C_VEL
LIN {X 0,Y 714.548,Z 1067.215,A -85,B 0,C 180,E1 26936.736,E2 26936.736} C_VEL
LIN {X 0,Y 713.971,Z 1085.45,A -85,B 0,C 180,E1 26935.108,E2 26935.108} C_VEL
LIN {X 0,Y 713.509,Z 1101.394,A -85,B 0,C 180,E1 26933.54,E2 26933.54} C_VEL
LIN {X 0,Y 713.048,Z 1120.126,A -85,B 0,C 180,E1 26931.468,E2 26931.468} C_VEL
LIN {X 0,Y 712.741,Z 1134.092,A -85,B 0,C 180,E1 26929.723,E2 26929.723} C_VEL
LIN {X 0,Y 712.498,Z 1146.004,A -85,B 0,C 180,E1 26928.067,E2 26928.067} C_VEL
LIN {X 0,Y 712.28,Z 1158.9,A -85,B 0,C 180,E1 26926.054,E2 26926.054} C_VEL
LIN {X 0,Y 712.124,Z 1170.245,A -85,B 0,C 180,E1 26923.975,E2 26923.975} C_VEL
LIN {X 0,Y 712.027,Z 1178.433,A -85,B 0,C 180,E1 26922.242,E2 26922.242} C_VEL
LIN {X 0,Y 711.979,Z 1186.134,A -85,B 0,C 180,E1 26920.356,E2 26920.356} C_VEL
LIN {X 0,Y 711.935,Z 1193.355,A -85,B 0,C 180,E1 26918.155,E2 26918.155} C_VEL
LIN {X 0,Y 711.916,Z 1198.765,A -85,B 0,C 180,E1 26915.965,E2 26915.965} C_VEL
LIN {X 0,Y 711.907,Z 1202.382,A -85,B 0,C 180,E1 26913.865,E2 26913.865} C_VEL
LIN {X 0,Y 711.909,Z 1204.549,A -85,B 0,C 180,E1 26911.609,E2 26911.609} C_VEL
LIN {X 0,Y 711.89,Z 1204.872,A -85,B 0,C 180,E1 26909.517,E2 26909.517} C_VEL
LIN {X 0,Y 711.907,Z 1203.967,A -85,B 0,C 180,E1 26907.585,E2 26907.585} C_VEL
LIN {X 0,Y 711.908,Z 1201.303,A -85,B 0,C 180,E1 26905.408,E2 26905.408} C_VEL
LIN {X 0,Y 711.919,Z 1197.151,A -85,B 0,C 180,E1 26903.306,E2 26903.306} C_VEL
LIN {X 0,Y 711.944,Z 1191.396,A -85,B 0,C 180,E1 26901.194,E2 26901.194} C_VEL
LIN {X 0,Y 711.976,Z 1183.956,A -85,B 0,C 180,E1 26899.071,E2 26899.071} C_VEL
LIN {X 0,Y 712.09,Z 1173.938,A -85,B 0,C 180,E1 26896.769,E2 26896.769} C_VEL
LIN {X 0,Y 712.178,Z 1164.528,A -85,B 0,C 180,E1 26894.946,E2 26894.946} C_VEL
LIN {X 0,Y 712.341,Z 1154.742,A -85,B 0,C 180,E1 26893.277,E2 26893.277} C_VEL
LIN {X 0,Y 712.541,Z 1143.674,A -85,B 0,C 180,E1 26891.595,E2 26891.595} C_VEL
LIN {X 0,Y 712.857,Z 1129.292,A -85,B 0,C 180,E1 26889.644,E2 26889.644} C_VEL
LIN {X 0,Y 713.224,Z 1112.619,A -85,B 0,C 180,E1 26887.671,E2 26887.671} C_VEL
LIN {X 0,Y 713.612,Z 1097.976,A -85,B 0,C 180,E1 26886.113,E2 26886.113} C_VEL
LIN {X 0,Y 714.175,Z 1079.334,A -85,B 0,C 180,E1 26884.317,E2 26884.317} C_VEL
LIN {X 0,Y 714.744,Z 1059.887,A -85,B 0,C 180,E1 26882.665,E2 26882.665} C_VEL
LIN {X 0,Y 715.326,Z 1042.229,A -85,B 0,C 180,E1 26881.305,E2 26881.305} C_VEL
LIN {X 0,Y 716.076,Z 1020.237,A -85,B 0,C 180,E1 26879.776,E2 26879.776} C_VEL
LIN {X 0,Y 716.773,Z 997.03,A -85,B 0,C 180,E1 26878.365,E2 26878.365} C_VEL
LIN {X 0,Y 717.452,Z 976.744,A -85,B 0,C 180,E1 26877.266,E2 26877.266} C_VEL
LIN {X 0,Y 718.178,Z 954.704,A -85,B 0,C 180,E1 26876.206,E2 26876.206} C_VEL
LIN {X 0,Y 718.923,Z 928.933,A -85,B 0,C 180,E1 26875.137,E2 26875.137} C_VEL
LIN {X 0,Y 719.505,Z 905.567,A -85,B 0,C 180,E1 26874.316,E2 26874.316} C_VEL
LIN {X 0,Y 720.071,Z 882.51,A -85,B 0,C 180,E1 26873.629,E2 26873.629} C_VEL
LIN {X 0,Y 720.651,Z 855.399,A -85,B 0,C 180,E1 26872.985,E2 26872.985} C_VEL
LIN {X 0,Y 721.044,Z 828.216,A -85,B 0,C 180,E1 26872.509,E2 26872.509} C_VEL
LIN {X 0,Y 722.49,Z 599.176,A -85,B 0,C 180,E1 26869.71,E2 26869.71} C_VEL
LIN {X 0,Y 723.793,Z 395.035,A -85,B 0,C 180,E1 26867.147,E2 26867.147} C_VEL
LIN {X 0,Y 723.858,Z 361.789,A -85,B 0,C 180,E1 26866.709,E2 26866.709} C_VEL
LIN {X 0,Y 721.092,Z 349.984,A -85,B 0,C 180,E1 26866.327,E2 26866.327} C_VEL
LIN {X 0,Y 721.275,Z 335.066,A -85,B 0,C 180,E1 26865.386,E2 26865.386} C_VEL
LIN {X 0,Y 715.838,Z 323.516,A -85,B 0,C 180,E1 26864.188,E2 26864.188} C_VEL
LIN {X 0,Y 712.28,Z 315.965,A -85,B 0,C 180,E1 26863.364,E2 26863.364} C_VEL
LIN {X 0,Y 712.245,Z 315.444,A -85,B 0,C 180,E1 26862.996,E2 26862.996} C_VEL
LIN {X 0,Y 712.206,Z 315.499,A -85,B 0,C 180,E1 26860.081,E2 26860.081} C_VEL
LIN {X 0,Y 712.196,Z 315.512,A -85,B 0,C 180,E1 26857.642,E2 26857.642} C_VEL
LIN {X 0,Y 712.236,Z 315.508,A -85,B 0,C 180,E1 26855.043,E2 26855.043} C_VEL
LIN {X 0,Y 712.224,Z 315.503,A -85,B 0,C 180,E1 26851.956,E2 26851.956} C_VEL
LIN {X 0,Y 712.21,Z 315.509,A -85,B 0,C 180,E1 26849.431,E2 26849.431} C_VEL
LIN {X 0,Y 712.274,Z 315.504,A -85,B 0,C 180,E1 26846.694,E2 26846.694} C_VEL
LIN {X 0,Y 712.23,Z 315.494,A -85,B 0,C 180,E1 26843.748,E2 26843.748} C_VEL
LIN {X 0,Y 712.23,Z 315.508,A -85,B 0,C 180,E1 26841.063,E2 26841.063} C_VEL
LIN {X 0,Y 712.279,Z 315.49,A -85,B 0,C 180,E1 26838.074,E2 26838.074} C_VEL
LIN {X 0,Y 712.228,Z 315.507,A -85,B 0,C 180,E1 26835.22,E2 26835.22} C_VEL
LIN {X 0,Y 712.279,Z 315.493,A -85,B 0,C 180,E1 26832.403,E2 26832.403} C_VEL
LIN {X 0,Y 712.245,Z 315.503,A -85,B 0,C 180,E1 26829.372,E2 26829.372} C_VEL
LIN {X 0,Y 712.276,Z 315.494,A -85,B 0,C 180,E1 26826.448,E2 26826.448} C_VEL
LIN {X 0,Y 712.262,Z 315.501,A -85,B 0,C 180,E1 26823.38,E2 26823.38} C_VEL
LIN {X 0,Y 712.274,Z 315.495,A -85,B 0,C 180,E1 26820.402,E2 26820.402} C_VEL
LIN {X 0,Y 712.269,Z 315.499,A -85,B 0,C 180,E1 26817.264,E2 26817.264} C_VEL
LIN {X 0,Y 712.276,Z 315.494,A -85,B 0,C 180,E1 26814.28,E2 26814.28} C_VEL
LIN {X 0,Y 712.278,Z 315.497,A -85,B 0,C 180,E1 26811.198,E2 26811.198} C_VEL
LIN {X 0,Y 712.273,Z 315.493,A -85,B 0,C 180,E1 26808.091,E2 26808.091} C_VEL
LIN {X 0,Y 712.279,Z 315.499,A -85,B 0,C 180,E1 26805.031,E2 26805.031} C_VEL
LIN {X 0,Y 712.272,Z 315.494,A -85,B 0,C 180,E1 26802.011,E2 26802.011} C_VEL
LIN {X 0,Y 712.275,Z 315.489,A -85,B 0,C 180,E1 26800.88,E2 26800.88} C_VEL
LIN {X 0,Y 711.29,Z 315.621,A -85,B 0,C 180,E1 26800.261,E2 26800.261} C_VEL
LIN {X 0,Y 704.894,Z 316.434,A -85,B 0,C 180,E1 26798.525,E2 26798.525} C_VEL
LIN {X 0,Y 704.342,Z 316.495,A -85,B 0,C 180,E1 26798.074,E2 26798.074} C_VEL
LIN {X 0,Y 704.318,Z 316.486,A -85,B 0,C 180,E1 26795.062,E2 26795.062} C_VEL
LIN {X 0,Y 704.339,Z 316.484,A -85,B 0,C 180,E1 26791.972,E2 26791.972} C_VEL
LIN {X 0,Y 704.307,Z 316.494,A -85,B 0,C 180,E1 26789.034,E2 26789.034} C_VEL
LIN {X 0,Y 704.339,Z 316.482,A -85,B 0,C 180,E1 26785.99,E2 26785.99} C_VEL
LIN {X 0,Y 704.29,Z 316.486,A -85,B 0,C 180,E1 26783.193,E2 26783.193} C_VEL
LIN {X 0,Y 704.344,Z 316.497,A -85,B 0,C 180,E1 26780.296,E2 26780.296} C_VEL
LIN {X 0,Y 704.291,Z 316.504,A -85,B 0,C 180,E1 26777.341,E2 26777.341} C_VEL
LIN {X 0,Y 704.358,Z 316.674,A -85,B 0,C 180,E1 26775.737,E2 26775.737} C_VEL
LIN {X 0,Y 705.654,Z 320.056,A -85,B 0,C 180,E1 26775.342,E2 26775.342} C_VEL
LIN {X 0,Y 711.796,Z 333.309,A -85,B 0,C 180,E1 26773.893,E2 26773.893} C_VEL
LIN {X 0,Y 714.046,Z 338.635,A -85,B 0,C 180,E1 26773.352,E2 26773.352} C_VEL
LIN {X 0,Y 712.908,Z 379.388,A -85,B 0,C 180,E1 26770.706,E2 26770.706} C_VEL
LIN {X 0,Y 712.629,Z 397.019,A -85,B 0,C 180,E1 26769.611,E2 26769.611} C_VEL
LIN {X 0,Y 715.523,Z 410.364,A -85,B 0,C 180,E1 26769.243,E2 26769.243} C_VEL
LIN {X 0,Y 713.917,Z 657.07,A -85,B 0,C 180,E1 26766.269,E2 26766.269} C_VEL
LIN {X 0,Y 712.792,Z 830.064,A -85,B 0,C 180,E1 26764.217,E2 26764.217} C_VEL
LIN {X 0,Y 712.427,Z 855.32,A -85,B 0,C 180,E1 26763.793,E2 26763.793} C_VEL
LIN {X 0,Y 711.812,Z 880.606,A -85,B 0,C 180,E1 26763.203,E2 26763.203} C_VEL
LIN {X 0,Y 711.287,Z 902.242,A -85,B 0,C 180,E1 26762.575,E2 26762.575} C_VEL
LIN {X 0,Y 710.608,Z 928.21,A -85,B 0,C 180,E1 26761.658,E2 26761.658} C_VEL
LIN {X 0,Y 709.865,Z 950.782,A -85,B 0,C 180,E1 26760.704,E2 26760.704} C_VEL
LIN {X 0,Y 709.127,Z 973.07,A -85,B 0,C 180,E1 26759.618,E2 26759.618} C_VEL
LIN {X 0,Y 708.343,Z 996.109,A -85,B 0,C 180,E1 26758.313,E2 26758.313} C_VEL
LIN {X 0,Y 707.67,Z 1014.909,A -85,B 0,C 180,E1 26757.108,E2 26757.108} C_VEL
LIN {X 0,Y 706.953,Z 1036.011,A -85,B 0,C 180,E1 26755.585,E2 26755.585} C_VEL
LIN {X 0,Y 706.355,Z 1053.548,A -85,B 0,C 180,E1 26754.148,E2 26754.148} C_VEL
LIN {X 0,Y 705.799,Z 1070.832,A -85,B 0,C 180,E1 26752.577,E2 26752.577} C_VEL
LIN {X 0,Y 705.293,Z 1088.414,A -85,B 0,C 180,E1 26750.758,E2 26750.758} C_VEL
LIN {X 0,Y 704.92,Z 1102.455,A -85,B 0,C 180,E1 26749.127,E2 26749.127} C_VEL
LIN {X 0,Y 704.57,Z 1117.89,A -85,B 0,C 180,E1 26747.083,E2 26747.083} C_VEL
LIN {X 0,Y 704.351,Z 1129.004,A -85,B 0,C 180,E1 26745.394,E2 26745.394} C_VEL
LIN {X 0,Y 704.183,Z 1139.21,A -85,B 0,C 180,E1 26743.633,E2 26743.633} C_VEL
LIN {X 0,Y 704.057,Z 1149.83,A -85,B 0,C 180,E1 26741.468,E2 26741.468} C_VEL
LIN {X 0,Y 703.962,Z 1157.073,A -85,B 0,C 180,E1 26739.686,E2 26739.686} C_VEL
LIN {X 0,Y 703.947,Z 1162.763,A -85,B 0,C 180,E1 26738.002,E2 26738.002} C_VEL
LIN {X 0,Y 703.911,Z 1168.279,A -85,B 0,C 180,E1 26735.952,E2 26735.952} C_VEL
LIN {X 0,Y 703.916,Z 1172.001,A -85,B 0,C 180,E1 26733.91,E2 26733.91} C_VEL
LIN {X 0,Y 703.914,Z 1173.968,A -85,B 0,C 180,E1 26732.198,E2 26732.198} C_VEL
LIN {X 0,Y 703.892,Z 1174.881,A -85,B 0,C 180,E1 26730.407,E2 26730.407} C_VEL
LIN {X 0,Y 703.906,Z 1174.379,A -85,B 0,C 180,E1 26728.209,E2 26728.209} C_VEL
LIN {X 0,Y 703.895,Z 1172.465,A -85,B 0,C 180,E1 26726.335,E2 26726.335} C_VEL
LIN {X 0,Y 703.911,Z 1169.595,A -85,B 0,C 180,E1 26724.621,E2 26724.621} C_VEL
LIN {X 0,Y 703.933,Z 1164.994,A -85,B 0,C 180,E1 26722.656,E2 26722.656} C_VEL
LIN {X 0,Y 703.972,Z 1158.458,A -85,B 0,C 180,E1 26720.599,E2 26720.599} C_VEL
LIN {X 0,Y 704.014,Z 1151.642,A -85,B 0,C 180,E1 26718.863,E2 26718.863} C_VEL
LIN {X 0,Y 704.124,Z 1143.969,A -85,B 0,C 180,E1 26717.202,E2 26717.202} C_VEL
LIN {X 0,Y 704.29,Z 1133.185,A -85,B 0,C 180,E1 26715.194,E2 26715.194} C_VEL
LIN {X 0,Y 704.51,Z 1120.83,A -85,B 0,C 180,E1 26713.255,E2 26713.255} C_VEL
LIN {X 0,Y 704.768,Z 1108.552,A -85,B 0,C 180,E1 26711.556,E2 26711.556} C_VEL
LIN {X 0,Y 705.171,Z 1092.329,A -85,B 0,C 180,E1 26709.586,E2 26709.586} C_VEL
LIN {X 0,Y 705.63,Z 1076.952,A -85,B 0,C 180,E1 26707.945,E2 26707.945} C_VEL
LIN {X 0,Y 706.192,Z 1058.641,A -85,B 0,C 180,E1 26706.202,E2 26706.202} C_VEL
LIN {X 0,Y 706.789,Z 1040.582,A -85,B 0,C 180,E1 26704.688,E2 26704.688} C_VEL
LIN {X 0,Y 707.488,Z 1020.816,A -85,B 0,C 180,E1 26703.203,E2 26703.203} C_VEL
LIN {X 0,Y 708.208,Z 999.734,A -85,B 0,C 180,E1 26701.819,E2 26701.819} C_VEL
LIN {X 0,Y 708.888,Z 980.514,A -85,B 0,C 180,E1 26700.697,E2 26700.697} C_VEL
LIN {X 0,Y 709.682,Z 956.679,A -85,B 0,C 180,E1 26699.475,E2 26699.475} C_VEL
LIN {X 0,Y 710.358,Z 934.878,A -85,B 0,C 180,E1 26698.52,E2 26698.52} C_VEL
LIN {X 0,Y 711.037,Z 912.845,A -85,B 0,C 180,E1 26697.689,E2 26697.689} C_VEL
LIN {X 0,Y 711.717,Z 887.082,A -85,B 0,C 180,E1 26696.882,E2 26696.882} C_VEL
LIN {X 0,Y 712.18,Z 864.23,A -85,B 0,C 180,E1 26696.31,E2 26696.31} C_VEL
LIN {X 0,Y 712.588,Z 841.639,A -85,B 0,C 180,E1 26695.868,E2 26695.868} C_VEL
LIN {X 0,Y 712.977,Z 809.028,A -85,B 0,C 180,E1 26695.426,E2 26695.426} C_VEL
LIN {X 0,Y 714.459,Z 570.522,A -85,B 0,C 180,E1 26692.608,E2 26692.608} C_VEL
LIN {X 0,Y 715.434,Z 409.066,A -85,B 0,C 180,E1 26690.645,E2 26690.645} C_VEL
LIN {X 0,Y 712.54,Z 396.176,A -85,B 0,C 180,E1 26690.264,E2 26690.264} C_VEL
LIN {X 0,Y 713.729,Z 350.042,A -85,B 0,C 180,E1 26687.309,E2 26687.309} C_VEL
LIN {X 0,Y 713.909,Z 338.098,A -85,B 0,C 180,E1 26686.511,E2 26686.511} C_VEL
LIN {X 0,Y 707.744,Z 324.412,A -85,B 0,C 180,E1 26685.057,E2 26685.057} C_VEL
LIN {X 0,Y 704.391,Z 316.924,A -85,B 0,C 180,E1 26684.22,E2 26684.22} C_VEL
LIN {X 0,Y 704.342,Z 316.475,A -85,B 0,C 180,E1 26683.963,E2 26683.963} C_VEL
LIN {X 0,Y 704.281,Z 316.48,A -85,B 0,C 180,E1 26681.074,E2 26681.074} C_VEL
LIN {X 0,Y 704.299,Z 316.496,A -85,B 0,C 180,E1 26678.403,E2 26678.403} C_VEL
LIN {X 0,Y 704.319,Z 316.495,A -85,B 0,C 180,E1 26675.285,E2 26675.285} C_VEL
LIN {X 0,Y 704.292,Z 316.486,A -85,B 0,C 180,E1 26672.511,E2 26672.511} C_VEL
LIN {X 0,Y 704.336,Z 316.48,A -85,B 0,C 180,E1 26669.606,E2 26669.606} C_VEL
LIN {X 0,Y 704.301,Z 316.494,A -85,B 0,C 180,E1 26666.747,E2 26666.747} C_VEL
LIN {X 0,Y 704.337,Z 316.481,A -85,B 0,C 180,E1 26663.866,E2 26663.866} C_VEL
LIN {X 0,Y 704.317,Z 316.492,A -85,B 0,C 180,E1 26660.788,E2 26660.788} C_VEL
LIN {X 0,Y 704.335,Z 316.481,A -85,B 0,C 180,E1 26657.857,E2 26657.857} C_VEL
LIN {X 0,Y 704.336,Z 316.488,A -85,B 0,C 180,E1 26654.805,E2 26654.805} C_VEL
LIN {X 0,Y 704.336,Z 316.482,A -85,B 0,C 180,E1 26651.713,E2 26651.713} C_VEL
LIN {X 0,Y 704.337,Z 316.487,A -85,B 0,C 180,E1 26648.655,E2 26648.655} C_VEL
LIN {X 0,Y 704.335,Z 316.482,A -85,B 0,C 180,E1 26645.621,E2 26645.621} C_VEL
LIN {X 0,Y 704.338,Z 316.488,A -85,B 0,C 180,E1 26642.522,E2 26642.522} C_VEL
LIN {X 0,Y 704.326,Z 316.484,A -85,B 0,C 180,E1 26639.431,E2 26639.431} C_VEL
LIN {X 0,Y 704.338,Z 316.489,A -85,B 0,C 180,E1 26636.419,E2 26636.419} C_VEL
LIN {X 0,Y 704.318,Z 316.485,A -85,B 0,C 180,E1 26633.315,E2 26633.315} C_VEL
LIN {X 0,Y 704.33,Z 316.489,A -85,B 0,C 180,E1 26630.356,E2 26630.356} C_VEL
LIN {X 0,Y 704.316,Z 316.486,A -85,B 0,C 180,E1 26627.237,E2 26627.237} C_VEL
LIN {X 0,Y 704.311,Z 316.492,A -85,B 0,C 180,E1 26624.351,E2 26624.351} C_VEL
LIN {X 0,Y 704.315,Z 316.489,A -85,B 0,C 180,E1 26621.2,E2 26621.2} C_VEL
LIN {X 0,Y 704.29,Z 316.493,A -85,B 0,C 180,E1 26618.419,E2 26618.419} C_VEL
LIN {X 0,Y 704.342,Z 316.487,A -85,B 0,C 180,E1 26615.421,E2 26615.421} C_VEL
LIN {X 0,Y 704.275,Z 316.488,A -85,B 0,C 180,E1 26612.613,E2 26612.613} C_VEL
LIN {X 0,Y 704.305,Z 316.495,A -85,B 0,C 180,E1 26609.924,E2 26609.924} C_VEL
LIN {X 0,Y 704.288,Z 316.491,A -85,B 0,C 180,E1 26606.866,E2 26606.866} C_VEL
LIN {X 0,Y 704.262,Z 316.495,A -85,B 0,C 180,E1 26604.301,E2 26604.301} C_VEL
LIN {X 0,Y 704.322,Z 316.499,A -85,B 0,C 180,E1 26601.552,E2 26601.552} C_VEL
LIN {X 0,Y 704.264,Z 316.507,A -85,B 0,C 180,E1 26598.558,E2 26598.558} C_VEL
LIN {X 0,Y 704.358,Z 316.661,A -85,B 0,C 180,E1 26597.303,E2 26597.303} C_VEL
LIN {X 0,Y 705.617,Z 319.937,A -85,B 0,C 180,E1 26596.92,E2 26596.92} C_VEL
LIN {X 0,Y 712.69,Z 334.443,A -85,B 0,C 180,E1 26595.34,E2 26595.34} C_VEL
LIN {X 0,Y 715.024,Z 339.584,A -85,B 0,C 180,E1 26594.812,E2 26594.812} C_VEL
LIN {X 0,Y 714.876,Z 350.757,A -85,B 0,C 180,E1 26594.127,E2 26594.127} C_VEL
LIN {X 0,Y 718.17,Z 365.32,A -85,B 0,C 180,E1 26593.672,E2 26593.672} C_VEL
LIN {X 0,Y 716.542,Z 577.719,A -85,B 0,C 180,E1 26590.973,E2 26590.973} C_VEL
LIN {X 0,Y 714.949,Z 802.518,A -85,B 0,C 180,E1 26588.211,E2 26588.211} C_VEL
LIN {X 0,Y 714.571,Z 836.319,A -85,B 0,C 180,E1 26587.758,E2 26587.758} C_VEL
LIN {X 0,Y 714.008,Z 863.287,A -85,B 0,C 180,E1 26587.233,E2 26587.233} C_VEL
LIN {X 0,Y 713.415,Z 888.48,A -85,B 0,C 180,E1 26586.593,E2 26586.593} C_VEL
LIN {X 0,Y 712.6,Z 916.838,A -85,B 0,C 180,E1 26585.686,E2 26585.686} C_VEL
LIN {X 0,Y 711.838,Z 939.491,A -85,B 0,C 180,E1 26584.819,E2 26584.819} C_VEL
LIN {X 0,Y 711.071,Z 960.698,A -85,B 0,C 180,E1 26583.886,E2 26583.886} C_VEL
LIN {X 0,Y 710.257,Z 982.228,A -85,B 0,C 180,E1 26582.812,E2 26582.812} C_VEL
LIN {X 0,Y 709.315,Z 1007.882,A -85,B 0,C 180,E1 26581.342,E2 26581.342} C_VEL
LIN {X 0,Y 708.531,Z 1027.572,A -85,B 0,C 180,E1 26580.064,E2 26580.064} C_VEL
LIN {X 0,Y 707.83,Z 1045.865,A -85,B 0,C 180,E1 26578.75,E2 26578.75} C_VEL
LIN {X 0,Y 707.057,Z 1066.708,A -85,B 0,C 180,E1 26577.087,E2 26577.087} C_VEL
LIN {X 0,Y 706.388,Z 1085.451,A -85,B 0,C 180,E1 26575.397,E2 26575.397} C_VEL
LIN {X 0,Y 705.819,Z 1101.773,A -85,B 0,C 180,E1 26573.773,E2 26573.773} C_VEL
LIN {X 0,Y 705.275,Z 1120.128,A -85,B 0,C 180,E1 26571.717,E2 26571.717} C_VEL
LIN {X 0,Y 704.919,Z 1133.809,A -85,B 0,C 180,E1 26569.989,E2 26569.989} C_VEL
LIN {X 0,Y 704.607,Z 1146.588,A -85,B 0,C 180,E1 26568.191,E2 26568.191} C_VEL
LIN {X 0,Y 704.335,Z 1160.068,A -85,B 0,C 180,E1 26566.036,E2 26566.036} C_VEL
LIN {X 0,Y 704.164,Z 1170.656,A -85,B 0,C 180,E1 26564.052,E2 26564.052} C_VEL
LIN {X 0,Y 704.053,Z 1178.792,A -85,B 0,C 180,E1 26562.3,E2 26562.3} C_VEL
LIN {X 0,Y 703.99,Z 1186.427,A -85,B 0,C 180,E1 26560.392,E2 26560.392} C_VEL
LIN {X 0,Y 703.94,Z 1193.595,A -85,B 0,C 180,E1 26558.166,E2 26558.166} C_VEL
LIN {X 0,Y 703.918,Z 1198.937,A -85,B 0,C 180,E1 26555.952,E2 26555.952} C_VEL
LIN {X 0,Y 703.908,Z 1202.484,A -85,B 0,C 180,E1 26553.828,E2 26553.828} C_VEL
LIN {X 0,Y 703.908,Z 1204.549,A -85,B 0,C 180,E1 26551.628,E2 26551.628} C_VEL
LIN {X 0,Y 703.89,Z 1204.872,A -85,B 0,C 180,E1 26549.511,E2 26549.511} C_VEL
LIN {X 0,Y 703.907,Z 1203.964,A -85,B 0,C 180,E1 26547.557,E2 26547.557} C_VEL
LIN {X 0,Y 703.909,Z 1201.428,A -85,B 0,C 180,E1 26545.437,E2 26545.437} C_VEL
LIN {X 0,Y 703.921,Z 1197.347,A -85,B 0,C 180,E1 26543.311,E2 26543.311} C_VEL
LIN {X 0,Y 703.949,Z 1191.393,A -85,B 0,C 180,E1 26541.093,E2 26541.093} C_VEL
LIN {X 0,Y 703.992,Z 1184.275,A -85,B 0,C 180,E1 26539.028,E2 26539.028} C_VEL
LIN {X 0,Y 704.128,Z 1173.939,A -85,B 0,C 180,E1 26536.617,E2 26536.617} C_VEL
LIN {X 0,Y 704.237,Z 1164.53,A -85,B 0,C 180,E1 26534.772,E2 26534.772} C_VEL
LIN {X 0,Y 704.437,Z 1154.7,A -85,B 0,C 180,E1 26533.076,E2 26533.076} C_VEL
LIN {X 0,Y 704.667,Z 1143.676,A -85,B 0,C 180,E1 26531.382,E2 26531.382} C_VEL
LIN {X 0,Y 705.06,Z 1128.615,A -85,B 0,C 180,E1 26529.322,E2 26529.322} C_VEL
LIN {X 0,Y 705.488,Z 1112.621,A -85,B 0,C 180,E1 26527.413,E2 26527.413} C_VEL
LIN {X 0,Y 705.994,Z 1097.124,A -85,B 0,C 180,E1 26525.75,E2 26525.75} C_VEL
LIN {X 0,Y 706.629,Z 1077.87,A -85,B 0,C 180,E1 26523.892,E2 26523.892} C_VEL
LIN {X 0,Y 707.336,Z 1059.05,A -85,B 0,C 180,E1 26522.285,E2 26522.285} C_VEL
LIN {X 0,Y 708.004,Z 1041.625,A -85,B 0,C 180,E1 26520.934,E2 26520.934} C_VEL
LIN {X 0,Y 708.863,Z 1019.175,A -85,B 0,C 180,E1 26519.366,E2 26519.366} C_VEL
LIN {X 0,Y 709.707,Z 997.005,A -85,B 0,C 180,E1 26518.011,E2 26518.011} C_VEL
LIN {X 0,Y 710.452,Z 977.637,A -85,B 0,C 180,E1 26516.951,E2 26516.951} C_VEL
LIN {X 0,Y 711.249,Z 956.609,A -85,B 0,C 180,E1 26515.924,E2 26515.924} C_VEL
LIN {X 0,Y 712.159,Z 930.744,A -85,B 0,C 180,E1 26514.827,E2 26514.827} C_VEL
LIN {X 0,Y 712.864,Z 906.304,A -85,B 0,C 180,E1 26513.956,E2 26513.956} C_VEL
LIN {X 0,Y 713.531,Z 883.182,A -85,B 0,C 180,E1 26513.261,E2 26513.261} C_VEL
LIN {X 0,Y 714.184,Z 856.721,A -85,B 0,C 180,E1 26512.624,E2 26512.624} C_VEL
LIN {X 0,Y 714.663,Z 829.442,A -85,B 0,C 180,E1 26512.135,E2 26512.135} C_VEL
LIN {X 0,Y 716.322,Z 607.037,A -85,B 0,C 180,E1 26509.392,E2 26509.392} C_VEL
LIN {X 0,Y 717.85,Z 403.688,A -85,B 0,C 180,E1 26506.821,E2 26506.821} C_VEL
LIN {X 0,Y 718.02,Z 363.911,A -85,B 0,C 180,E1 26506.297,E2 26506.297} C_VEL
LIN {X 0,Y 714.767,Z 349.995,A -85,B 0,C 180,E1 26505.841,E2 26505.841} C_VEL
LIN {X 0,Y 714.916,Z 339.314,A -85,B 0,C 180,E1 26505.162,E2 26505.162} C_VEL
LIN {X 0,Y 708.254,Z 325.058,A -85,B 0,C 180,E1 26503.658,E2 26503.658} C_VEL
LIN {X 0,Y 704.457,Z 317.18,A -85,B 0,C 180,E1 26502.779,E2 26502.779} C_VEL
LIN {X 0,Y 704.337,Z 316.567,A -85,B 0,C 180,E1 26502.622,E2 26502.622} C_VEL
LIN {X 0,Y 704.253,Z 316.488,A -85,B 0,C 180,E1 26499.816,E2 26499.816} C_VEL
LIN {X 0,Y 704.263,Z 316.498,A -85,B 0,C 180,E1 26497.421,E2 26497.421} C_VEL
LIN {X 0,Y 704.341,Z 316.496,A -85,B 0,C 180,E1 26494.502,E2 26494.502} C_VEL
LIN {X 0,Y 704.268,Z 316.493,A -85,B 0,C 180,E1 26491.689,E2 26491.689} C_VEL
LIN {X 0,Y 704.285,Z 316.498,A -85,B 0,C 180,E1 26489.141,E2 26489.141} C_VEL
LIN {X 0,Y 704.325,Z 316.494,A -85,B 0,C 180,E1 26486.11,E2 26486.11} C_VEL
LIN {X 0,Y 704.278,Z 316.484,A -85,B 0,C 180,E1 26483.335,E2 26483.335} C_VEL
LIN {X 0,Y 704.344,Z 316.498,A -85,B 0,C 180,E1 26480.527,E2 26480.527} C_VEL
LIN {X 0,Y 704.293,Z 316.48,A -85,B 0,C 180,E1 26477.516,E2 26477.516} C_VEL
LIN {X 0,Y 704.316,Z 316.5,A -85,B 0,C 180,E1 26474.721,E2 26474.721} C_VEL
LIN {X 0,Y 704.317,Z 316.479,A -85,B 0,C 180,E1 26471.606,E2 26471.606} C_VEL
LIN {X 0,Y 704.313,Z 316.498,A -85,B 0,C 180,E1 26468.737,E2 26468.737} C_VEL
LIN {X 0,Y 704.338,Z 316.477,A -85,B 0,C 180,E1 26465.651,E2 26465.651} C_VEL
LIN {X 0,Y 704.316,Z 316.498,A -85,B 0,C 180,E1 26462.685,E2 26462.685} C_VEL
LIN {X 0,Y 704.334,Z 316.475,A -85,B 0,C 180,E1 26459.675,E2 26459.675} C_VEL
LIN {X 0,Y 704.314,Z 316.494,A -85,B 0,C 180,E1 26456.745,E2 26456.745} C_VEL
LIN {X 0,Y 704.324,Z 316.476,A -85,B 0,C 180,E1 26453.888,E2 26453.888} C_VEL
LIN {X 0,Y 704.323,Z 316.489,A -85,B 0,C 180,E1 26450.933,E2 26450.933} C_VEL
LIN {X 0,Y 704.325,Z 316.478,A -85,B 0,C 180,E1 26447.954,E2 26447.954} C_VEL
LIN {X 0,Y 704.336,Z 316.489,A -85,B 0,C 180,E1 26444.942,E2 26444.942} C_VEL
LIN {X 0,Y 704.323,Z 316.48,A -85,B 0,C 180,E1 26441.886,E2 26441.886} C_VEL
LIN {X 0,Y 704.343,Z 316.489,A -85,B 0,C 180,E1 26438.855,E2 26438.855} C_VEL
LIN {X 0,Y 704.342,Z 316.495,A -85,B 0,C 180,E1 26438.074,E2 26438.074} C_VEL
LIN {X 0,Y 703.321,Z 316.611,A -85,B 0,C 180,E1 26437.447,E2 26437.447} C_VEL
LIN {X 0,Y 696.885,Z 317.413,A -85,B 0,C 180,E1 26435.692,E2 26435.692} C_VEL
LIN {X 0,Y 696.369,Z 317.476,A -85,B 0,C 180,E1 26435.236,E2 26435.236} C_VEL
LIN {X 0,Y 696.397,Z 317.479,A -85,B 0,C 180,E1 26432.277,E2 26432.277} C_VEL
LIN {X 0,Y 696.363,Z 317.488,A -85,B 0,C 180,E1 26429.449,E2 26429.449} C_VEL
LIN {X 0,Y 696.401,Z 317.464,A -85,B 0,C 180,E1 26426.532,E2 26426.532} C_VEL
LIN {X 0,Y 696.364,Z 317.476,A -85,B 0,C 180,E1 26423.522,E2 26423.522} C_VEL
LIN {X 0,Y 696.37,Z 317.487,A -85,B 0,C 180,E1 26420.707,E2 26420.707} C_VEL
LIN {X 0,Y 696.37,Z 317.487,A -85,B 0,C 180,E1 26417.557,E2 26417.557} C_VEL
LIN {X 0,Y 696.421,Z 317.679,A -85,B 0,C 180,E1 26416.354,E2 26416.354} C_VEL
LIN {X 0,Y 697.677,Z 320.899,A -85,B 0,C 180,E1 26415.965,E2 26415.965} C_VEL
LIN {X 0,Y 705.494,Z 337.589,A -85,B 0,C 180,E1 26414.098,E2 26414.098} C_VEL
LIN {X 0,Y 707.536,Z 342.809,A -85,B 0,C 180,E1 26413.566,E2 26413.566} C_VEL
LIN {X 0,Y 706.21,Z 384.244,A -85,B 0,C 180,E1 26410.853,E2 26410.853} C_VEL
LIN {X 0,Y 705.932,Z 396.577,A -85,B 0,C 180,E1 26410.073,E2 26410.073} C_VEL
LIN {X 0,Y 709.309,Z 412.182,A -85,B 0,C 180,E1 26409.632,E2 26409.632} C_VEL
LIN {X 0,Y 707.458,Z 658.138,A -85,B 0,C 180,E1 26406.642,E2 26406.642} C_VEL
LIN {X 0,Y 706.169,Z 830.108,A -85,B 0,C 180,E1 26404.584,E2 26404.584} C_VEL
LIN {X 0,Y 705.74,Z 855.625,A -85,B 0,C 180,E1 26404.15,E2 26404.15} C_VEL
LIN {X 0,Y 705.07,Z 880.516,A -85,B 0,C 180,E1 26403.566,E2 26403.566} C_VEL
LIN {X 0,Y 704.448,Z 902.264,A -85,B 0,C 180,E1 26402.931,E2 26402.931} C_VEL
LIN {X 0,Y 703.664,Z 928.22,A -85,B 0,C 180,E1 26402.007,E2 26402.007} C_VEL
LIN {X 0,Y 702.867,Z 949.925,A -85,B 0,C 180,E1 26401.085,E2 26401.085} C_VEL
LIN {X 0,Y 702.068,Z 970.417,A -85,B 0,C 180,E1 26400.087,E2 26400.087} C_VEL
LIN {X 0,Y 701.117,Z 994.646,A -85,B 0,C 180,E1 26398.725,E2 26398.725} C_VEL
LIN {X 0,Y 700.353,Z 1013.593,A -85,B 0,C 180,E1 26397.507,E2 26397.507} C_VEL
LIN {X 0,Y 699.533,Z 1034.15,A -85,B 0,C 180,E1 26396.028,E2 26396.028} C_VEL
LIN {X 0,Y 698.762,Z 1053.554,A -85,B 0,C 180,E1 26394.427,E2 26394.427} C_VEL
LIN {X 0,Y 698.147,Z 1070.374,A -85,B 0,C 180,E1 26392.882,E2 26392.882} C_VEL
LIN {X 0,Y 697.563,Z 1087.805,A -85,B 0,C 180,E1 26391.069,E2 26391.069} C_VEL
LIN {X 0,Y 697.115,Z 1101.753,A -85,B 0,C 180,E1 26389.436,E2 26389.436} C_VEL
LIN {X 0,Y 696.716,Z 1116.734,A -85,B 0,C 180,E1 26387.454,E2 26387.454} C_VEL
LIN {X 0,Y 696.432,Z 1129.009,A -85,B 0,C 180,E1 26385.574,E2 26385.574} C_VEL
LIN {X 0,Y 696.226,Z 1139.211,A -85,B 0,C 180,E1 26383.792,E2 26383.792} C_VEL
LIN {X 0,Y 696.082,Z 1149.951,A -85,B 0,C 180,E1 26381.574,E2 26381.574} C_VEL
LIN {X 0,Y 695.976,Z 1156.907,A -85,B 0,C 180,E1 26379.844,E2 26379.844} C_VEL
LIN {X 0,Y 695.954,Z 1162.599,A -85,B 0,C 180,E1 26378.148,E2 26378.148} C_VEL
LIN {X 0,Y 695.928,Z 1167.867,A -85,B 0,C 180,E1 26376.186,E2 26376.186} C_VEL
LIN {X 0,Y 695.917,Z 1171.889,A -85,B 0,C 180,E1 26374.037,E2 26374.037} C_VEL
LIN {X 0,Y 695.914,Z 1173.968,A -85,B 0,C 180,E1 26372.223,E2 26372.223} C_VEL
LIN {X 0,Y 695.891,Z 1174.881,A -85,B 0,C 180,E1 26370.412,E2 26370.412} C_VEL
LIN {X 0,Y 695.907,Z 1174.379,A -85,B 0,C 180,E1 26368.189,E2 26368.189} C_VEL
LIN {X 0,Y 695.898,Z 1172.464,A -85,B 0,C 180,E1 26366.293,E2 26366.293} C_VEL
LIN {X 0,Y 695.908,Z 1169.594,A -85,B 0,C 180,E1 26364.559,E2 26364.559} C_VEL
LIN {X 0,Y 695.935,Z 1165.2,A -85,B 0,C 180,E1 26362.654,E2 26362.654} C_VEL
LIN {X 0,Y 695.976,Z 1158.457,A -85,B 0,C 180,E1 26360.49,E2 26360.49} C_VEL
LIN {X 0,Y 696.042,Z 1151.641,A -85,B 0,C 180,E1 26358.734,E2 26358.734} C_VEL
LIN {X 0,Y 696.167,Z 1143.558,A -85,B 0,C 180,E1 26356.968,E2 26356.968} C_VEL
LIN {X 0,Y 696.361,Z 1132.15,A -85,B 0,C 180,E1 26354.851,E2 26354.851} C_VEL
LIN {X 0,Y 696.615,Z 1120.828,A -85,B 0,C 180,E1 26353.06,E2 26353.06} C_VEL
LIN {X 0,Y 696.922,Z 1108.55,A -85,B 0,C 180,E1 26351.341,E2 26351.341} C_VEL
LIN {X 0,Y 697.395,Z 1092.322,A -85,B 0,C 180,E1 26349.348,E2 26349.348} C_VEL
LIN {X 0,Y 697.904,Z 1077.536,A -85,B 0,C 180,E1 26347.749,E2 26347.749} C_VEL
LIN {X 0,Y 698.55,Z 1059.648,A -85,B 0,C 180,E1 26346.015,E2 26346.015} C_VEL
LIN {X 0,Y 699.261,Z 1040.821,A -85,B 0,C 180,E1 26344.416,E2 26344.416} C_VEL
LIN {X 0,Y 700.04,Z 1021.415,A -85,B 0,C 180,E1 26342.941,E2 26342.941} C_VEL
LIN {X 0,Y 700.921,Z 999.613,A -85,B 0,C 180,E1 26341.492,E2 26341.492} C_VEL
LIN {X 0,Y 701.692,Z 980.5,A -85,B 0,C 180,E1 26340.366,E2 26340.366} C_VEL
LIN {X 0,Y 702.607,Z 956.571,A -85,B 0,C 180,E1 26339.13,E2 26339.13} C_VEL
LIN {X 0,Y 703.401,Z 934.869,A -85,B 0,C 180,E1 26338.172,E2 26338.172} C_VEL
LIN {X 0,Y 704.156,Z 913.114,A -85,B 0,C 180,E1 26337.345,E2 26337.345} C_VEL
LIN {X 0,Y 704.928,Z 887.409,A -85,B 0,C 180,E1 26336.531,E2 26336.531} C_VEL
LIN {X 0,Y 705.469,Z 864.206,A -85,B 0,C 180,E1 26335.946,E2 26335.946} C_VEL
LIN {X 0,Y 705.95,Z 841.557,A -85,B 0,C 180,E1 26335.501,E2 26335.501} C_VEL
LIN {X 0,Y 706.383,Z 808.837,A -85,B 0,C 180,E1 26335.055,E2 26335.055} C_VEL
LIN {X 0,Y 708.091,Z 570.674,A -85,B 0,C 180,E1 26332.216,E2 26332.216} C_VEL
LIN {X 0,Y 709.238,Z 410.97,A -85,B 0,C 180,E1 26330.258,E2 26330.258} C_VEL
LIN {X 0,Y 705.927,Z 396.484,A -85,B 0,C 180,E1 26329.833,E2 26329.833} C_VEL
LIN {X 0,Y 707.266,Z 350.839,A -85,B 0,C 180,E1 26326.88,E2 26326.88} C_VEL
LIN {X 0,Y 707.383,Z 342.005,A -85,B 0,C 180,E1 26326.275,E2 26326.275} C_VEL
LIN {X 0,Y 701.51,Z 329.091,A -85,B 0,C 180,E1 26324.874,E2 26324.874} C_VEL
LIN {X 0,Y 697.592,Z 320.767,A -85,B 0,C 180,E1 26323.927,E2 26323.927} C_VEL
LIN {X 0,Y 696.402,Z 317.642,A -85,B 0,C 180,E1 26323.544,E2 26323.544} C_VEL
LIN {X 0,Y 696.338,Z 317.468,A -85,B 0,C 180,E1 26320.795,E2 26320.795} C_VEL
LIN {X 0,Y 696.403,Z 317.468,A -85,B 0,C 180,E1 26317.979,E2 26317.979} C_VEL
LIN {X 0,Y 696.36,Z 317.486,A -85,B 0,C 180,E1 26315.055,E2 26315.055} C_VEL
LIN {X 0,Y 696.37,Z 317.476,A -85,B 0,C 180,E1 26312.252,E2 26312.252} C_VEL
LIN {X 0,Y 696.382,Z 317.464,A -85,B 0,C 180,E1 26309.127,E2 26309.127} C_VEL
LIN {X 0,Y 696.377,Z 317.488,A -85,B 0,C 180,E1 26306.183,E2 26306.183} C_VEL
LIN {X 0,Y 696.392,Z 317.471,A -85,B 0,C 180,E1 26303.024,E2 26303.024} C_VEL
LIN {X 0,Y 696.385,Z 317.485,A -85,B 0,C 180,E1 26300.07,E2 26300.07} C_VEL
LIN {X 0,Y 696.399,Z 317.474,A -85,B 0,C 180,E1 26296.946,E2 26296.946} C_VEL
LIN {X 0,Y 696.397,Z 317.475,A -85,B 0,C 180,E1 26293.874,E2 26293.874} C_VEL
LIN {X 0,Y 696.399,Z 317.474,A -85,B 0,C 180,E1 26290.758,E2 26290.758} C_VEL
LIN {X 0,Y 696.399,Z 317.47,A -85,B 0,C 180,E1 26287.674,E2 26287.674} C_VEL
LIN {X 0,Y 696.399,Z 317.473,A -85,B 0,C 180,E1 26284.529,E2 26284.529} C_VEL
LIN {X 0,Y 696.389,Z 317.471,A -85,B 0,C 180,E1 26281.481,E2 26281.481} C_VEL
LIN {X 0,Y 696.401,Z 317.472,A -85,B 0,C 180,E1 26278.437,E2 26278.437} C_VEL
LIN {X 0,Y 696.386,Z 317.474,A -85,B 0,C 180,E1 26275.388,E2 26275.388} C_VEL
LIN {X 0,Y 696.392,Z 317.471,A -85,B 0,C 180,E1 26272.409,E2 26272.409} C_VEL
LIN {X 0,Y 696.384,Z 317.475,A -85,B 0,C 180,E1 26269.326,E2 26269.326} C_VEL
LIN {X 0,Y 696.375,Z 317.475,A -85,B 0,C 180,E1 26266.38,E2 26266.38} C_VEL
LIN {X 0,Y 696.375,Z 317.473,A -85,B 0,C 180,E1 26263.225,E2 26263.225} C_VEL
LIN {X 0,Y 696.359,Z 317.48,A -85,B 0,C 180,E1 26260.367,E2 26260.367} C_VEL
LIN {X 0,Y 696.4,Z 317.469,A -85,B 0,C 180,E1 26257.369,E2 26257.369} C_VEL
LIN {X 0,Y 696.34,Z 317.487,A -85,B 0,C 180,E1 26254.574,E2 26254.574} C_VEL
LIN {X 0,Y 696.388,Z 317.467,A -85,B 0,C 180,E1 26251.811,E2 26251.811} C_VEL
LIN {X 0,Y 696.343,Z 317.483,A -85,B 0,C 180,E1 26248.777,E2 26248.777} C_VEL
LIN {X 0,Y 696.33,Z 317.486,A -85,B 0,C 180,E1 26246.24,E2 26246.24} C_VEL
LIN {X 0,Y 696.404,Z 317.466,A -85,B 0,C 180,E1 26243.324,E2 26243.324} C_VEL
LIN {X 0,Y 696.318,Z 317.477,A -85,B 0,C 180,E1 26240.453,E2 26240.453} C_VEL
LIN {X 0,Y 696.328,Z 317.557,A -85,B 0,C 180,E1 26237.998,E2 26237.998} C_VEL
LIN {X 0,Y 696.619,Z 318.817,A -85,B 0,C 180,E1 26237.798,E2 26237.798} C_VEL
LIN {X 0,Y 698.822,Z 323.099,A -85,B 0,C 180,E1 26237.296,E2 26237.296} C_VEL
LIN {X 0,Y 707.292,Z 340.685,A -85,B 0,C 180,E1 26235.363,E2 26235.363} C_VEL
LIN {X 0,Y 708.649,Z 343.793,A -85,B 0,C 180,E1 26235.045,E2 26235.045} C_VEL
LIN {X 0,Y 708.617,Z 350.882,A -85,B 0,C 180,E1 26234.618,E2 26234.618} C_VEL
LIN {X 0,Y 712.354,Z 367.331,A -85,B 0,C 180,E1 26234.093,E2 26234.093} C_VEL
LIN {X 0,Y 710.478,Z 579.426,A -85,B 0,C 180,E1 26231.376,E2 26231.376} C_VEL
LIN {X 0,Y 708.646,Z 803.959,A -85,B 0,C 180,E1 26228.595,E2 26228.595} C_VEL
LIN {X 0,Y 708.211,Z 836.923,A -85,B 0,C 180,E1 26228.146,E2 26228.146} C_VEL
LIN {X 0,Y 707.577,Z 863.553,A -85,B 0,C 180,E1 26227.622,E2 26227.622} C_VEL
LIN {X 0,Y 706.897,Z 888.666,A -85,B 0,C 180,E1 26226.98,E2 26226.98} C_VEL
LIN {X 0,Y 705.969,Z 916.891,A -85,B 0,C 180,E1 26226.072,E2 26226.072} C_VEL
LIN {X 0,Y 705.112,Z 939.378,A -85,B 0,C 180,E1 26225.205,E2 26225.205} C_VEL
LIN {X 0,Y 704.279,Z 959.707,A -85,B 0,C 180,E1 26224.307,E2 26224.307} C_VEL
LIN {X 0,Y 703.406,Z 979.973,A -85,B 0,C 180,E1 26223.296,E2 26223.296} C_VEL
LIN {X 0,Y 702.349,Z 1004.205,A -85,B 0,C 180,E1 26221.929,E2 26221.929} C_VEL
LIN {X 0,Y 701.361,Z 1026.249,A -85,B 0,C 180,E1 26220.499,E2 26220.499} C_VEL
LIN {X 0,Y 700.541,Z 1044.716,A -85,B 0,C 180,E1 26219.166,E2 26219.166} C_VEL
LIN {X 0,Y 699.646,Z 1065.145,A -85,B 0,C 180,E1 26217.537,E2 26217.537} C_VEL
LIN {X 0,Y 698.842,Z 1084.52,A -85,B 0,C 180,E1 26215.782,E2 26215.782} C_VEL
LIN {X 0,Y 698.206,Z 1100.543,A -85,B 0,C 180,E1 26214.178,E2 26214.178} C_VEL
LIN {X 0,Y 697.592,Z 1118.364,A -85,B 0,C 180,E1 26212.189,E2 26212.189} C_VEL
LIN {X 0,Y 697.091,Z 1133.811,A -85,B 0,C 180,E1 26210.223,E2 26210.223} C_VEL
LIN {X 0,Y 696.732,Z 1146.59,A -85,B 0,C 180,E1 26208.404,E2 26208.404} C_VEL
LIN {X 0,Y 696.411,Z 1159.878,A -85,B 0,C 180,E1 26206.258,E2 26206.258} C_VEL
LIN {X 0,Y 696.215,Z 1170.714,A -85,B 0,C 180,E1 26204.204,E2 26204.204} C_VEL
LIN {X 0,Y 696.087,Z 1178.793,A -85,B 0,C 180,E1 26202.443,E2 26202.443} C_VEL
LIN {X 0,Y 695.998,Z 1186.427,A -85,B 0,C 180,E1 26200.512,E2 26200.512} C_VEL
LIN {X 0,Y 695.949,Z 1193.595,A -85,B 0,C 180,E1 26198.26,E2 26198.26} C_VEL
LIN {X 0,Y 695.92,Z 1198.937,A -85,B 0,C 180,E1 26196.02,E2 26196.02} C_VEL
LIN {X 0,Y 695.908,Z 1202.484,A -85,B 0,C 180,E1 26193.872,E2 26193.872} C_VEL
LIN {X 0,Y 695.908,Z 1204.549,A -85,B 0,C 180,E1 26191.646,E2 26191.646} C_VEL
LIN {X 0,Y 695.89,Z 1204.872,A -85,B 0,C 180,E1 26189.506,E2 26189.506} C_VEL
LIN {X 0,Y 695.907,Z 1203.961,A -85,B 0,C 180,E1 26187.529,E2 26187.529} C_VEL
LIN {X 0,Y 695.909,Z 1201.427,A -85,B 0,C 180,E1 26185.385,E2 26185.385} C_VEL
LIN {X 0,Y 695.923,Z 1197.347,A -85,B 0,C 180,E1 26183.234,E2 26183.234} C_VEL
LIN {X 0,Y 695.957,Z 1191.39,A -85,B 0,C 180,E1 26180.99,E2 26180.99} C_VEL
LIN {X 0,Y 696.017,Z 1184.162,A -85,B 0,C 180,E1 26178.871,E2 26178.871} C_VEL
LIN {X 0,Y 696.165,Z 1173.938,A -85,B 0,C 180,E1 26176.461,E2 26176.461} C_VEL
LIN {X 0,Y 696.308,Z 1164.532,A -85,B 0,C 180,E1 26174.594,E2 26174.594} C_VEL
LIN {X 0,Y 696.535,Z 1154.745,A -85,B 0,C 180,E1 26172.886,E2 26172.886} C_VEL
LIN {X 0,Y 696.809,Z 1143.678,A -85,B 0,C 180,E1 26171.164,E2 26171.164} C_VEL
LIN {X 0,Y 697.256,Z 1128.613,A -85,B 0,C 180,E1 26169.079,E2 26169.079} C_VEL
LIN {X 0,Y 697.77,Z 1112.485,A -85,B 0,C 180,E1 26167.133,E2 26167.133} C_VEL
LIN {X 0,Y 698.355,Z 1097.125,A -85,B 0,C 180,E1 26165.467,E2 26165.467} C_VEL
LIN {X 0,Y 699.102,Z 1077.869,A -85,B 0,C 180,E1 26163.589,E2 26163.589} C_VEL
LIN {X 0,Y 699.907,Z 1059.05,A -85,B 0,C 180,E1 26161.965,E2 26161.965} C_VEL
LIN {X 0,Y 700.676,Z 1041.626,A -85,B 0,C 180,E1 26160.6,E2 26160.6} C_VEL
LIN {X 0,Y 701.655,Z 1019.529,A -85,B 0,C 180,E1 26159.04,E2 26159.04} C_VEL
LIN {X 0,Y 702.662,Z 997.034,A -85,B 0,C 180,E1 26157.653,E2 26157.653} C_VEL
LIN {X 0,Y 703.514,Z 977.639,A -85,B 0,C 180,E1 26156.582,E2 26156.582} C_VEL
LIN {X 0,Y 704.373,Z 957.711,A -85,B 0,C 180,E1 26155.599,E2 26155.599} C_VEL
LIN {X 0,Y 705.355,Z 933.831,A -85,B 0,C 180,E1 26154.565,E2 26154.565} C_VEL
LIN {X 0,Y 706.254,Z 907.039,A -85,B 0,C 180,E1 26153.59,E2 26153.59} C_VEL
LIN {X 0,Y 707.028,Z 883.658,A -85,B 0,C 180,E1 26152.881,E2 26152.881} C_VEL
LIN {X 0,Y 707.752,Z 857.811,A -85,B 0,C 180,E1 26152.251,E2 26152.251} C_VEL
LIN {X 0,Y 708.318,Z 830.235,A -85,B 0,C 180,E1 26151.747,E2 26151.747} C_VEL
LIN {X 0,Y 709.236,Z 729.037,A -85,B 0,C 180,E1 26150.486,E2 26150.486} C_VEL
LIN {X 0,Y 711.104,Z 507.897,A -85,B 0,C 180,E1 26147.719,E2 26147.719} C_VEL
LIN {X 0,Y 712.208,Z 365.976,A -85,B 0,C 180,E1 26145.877,E2 26145.877} C_VEL
LIN {X 0,Y 708.486,Z 349.913,A -85,B 0,C 180,E1 26145.341,E2 26145.341} C_VEL
LIN {X 0,Y 708.593,Z 343.502,A -85,B 0,C 180,E1 26144.931,E2 26144.931} C_VEL
LIN {X 0,Y 701.772,Z 329.28,A -85,B 0,C 180,E1 26143.394,E2 26143.394} C_VEL
LIN {X 0,Y 698.125,Z 321.569,A -85,B 0,C 180,E1 26142.534,E2 26142.534} C_VEL
LIN {X 0,Y 696.399,Z 317.965,A -85,B 0,C 180,E1 26142.107,E2 26142.107} C_VEL
LIN {X 0,Y 696.311,Z 317.482,A -85,B 0,C 180,E1 26141.818,E2 26141.818} C_VEL
LIN {X 0,Y 696.325,Z 317.478,A -85,B 0,C 180,E1 26139.397,E2 26139.397} C_VEL
LIN {X 0,Y 696.391,Z 317.468,A -85,B 0,C 180,E1 26136.472,E2 26136.472} C_VEL
LIN {X 0,Y 696.326,Z 317.487,A -85,B 0,C 180,E1 26133.661,E2 26133.661} C_VEL
LIN {X 0,Y 696.362,Z 317.484,A -85,B 0,C 180,E1 26130.995,E2 26130.995} C_VEL
LIN {X 0,Y 696.355,Z 317.473,A -85,B 0,C 180,E1 26127.911,E2 26127.911} C_VEL
LIN {X 0,Y 696.343,Z 317.489,A -85,B 0,C 180,E1 26125.228,E2 26125.228} C_VEL
LIN {X 0,Y 696.405,Z 317.476,A -85,B 0,C 180,E1 26122.275,E2 26122.275} C_VEL
LIN {X 0,Y 696.347,Z 317.482,A -85,B 0,C 180,E1 26119.372,E2 26119.372} C_VEL
LIN {X 0,Y 696.4,Z 317.476,A -85,B 0,C 180,E1 26116.516,E2 26116.516} C_VEL
LIN {X 0,Y 696.369,Z 317.475,A -85,B 0,C 180,E1 26113.535,E2 26113.535} C_VEL
LIN {X 0,Y 696.378,Z 317.475,A -85,B 0,C 180,E1 26110.674,E2 26110.674} C_VEL
LIN {X 0,Y 696.382,Z 317.472,A -85,B 0,C 180,E1 26107.508,E2 26107.508} C_VEL
LIN {X 0,Y 696.388,Z 317.475,A -85,B 0,C 180,E1 26104.529,E2 26104.529} C_VEL
LIN {X 0,Y 696.391,Z 317.473,A -85,B 0,C 180,E1 26101.399,E2 26101.399} C_VEL
LIN {X 0,Y 696.398,Z 317.473,A -85,B 0,C 180,E1 26098.354,E2 26098.354} C_VEL
LIN {X 0,Y 696.392,Z 317.474,A -85,B 0,C 180,E1 26095.223,E2 26095.223} C_VEL
LIN {X 0,Y 696.4,Z 317.473,A -85,B 0,C 180,E1 26092.16,E2 26092.16} C_VEL
LIN {X 0,Y 696.396,Z 317.474,A -85,B 0,C 180,E1 26089.075,E2 26089.075} C_VEL
LIN {X 0,Y 696.395,Z 317.476,A -85,B 0,C 180,E1 26086.042,E2 26086.042} C_VEL
LIN {X 0,Y 696.4,Z 317.474,A -85,B 0,C 180,E1 26082.968,E2 26082.968} C_VEL
LIN {X 0,Y 696.386,Z 317.484,A -85,B 0,C 180,E1 26079.888,E2 26079.888} C_VEL
LIN {X 0,Y 696.401,Z 317.47,A -85,B 0,C 180,E1 26076.833,E2 26076.833} C_VEL
LIN {X 0,Y 696.369,Z 317.476,A -85,B 0,C 180,E1 26075.236,E2 26075.236} C_VEL
LIN {X 0,Y 695.405,Z 317.599,A -85,B 0,C 180,E1 26074.602,E2 26074.602} C_VEL
LIN {X 0,Y 689,Z 318.411,A -85,B 0,C 180,E1 26072.826,E2 26072.826} C_VEL
LIN {X 0,Y 688.459,Z 318.468,A -85,B 0,C 180,E1 26072.364,E2 26072.364} C_VEL
LIN {X 0,Y 688.424,Z 318.477,A -85,B 0,C 180,E1 26069.446,E2 26069.446} C_VEL
LIN {X 0,Y 688.463,Z 318.451,A -85,B 0,C 180,E1 26066.475,E2 26066.475} C_VEL
LIN {X 0,Y 688.42,Z 318.464,A -85,B 0,C 180,E1 26063.451,E2 26063.451} C_VEL
LIN {X 0,Y 688.442,Z 318.476,A -85,B 0,C 180,E1 26060.594,E2 26060.594} C_VEL
LIN {X 0,Y 688.427,Z 318.476,A -85,B 0,C 180,E1 26057.516,E2 26057.516} C_VEL
LIN {X 0,Y 688.465,Z 318.871,A -85,B 0,C 180,E1 26056.962,E2 26056.962} C_VEL
LIN {X 0,Y 690.146,Z 322.508,A -85,B 0,C 180,E1 26056.513,E2 26056.513} C_VEL
LIN {X 0,Y 699.446,Z 342.566,A -85,B 0,C 180,E1 26054.236,E2 26054.236} C_VEL
LIN {X 0,Y 701.081,Z 346.697,A -85,B 0,C 180,E1 26053.808,E2 26053.808} C_VEL
LIN {X 0,Y 699.537,Z 388.293,A -85,B 0,C 180,E1 26051.055,E2 26051.055} C_VEL
LIN {X 0,Y 699.42,Z 397.043,A -85,B 0,C 180,E1 26050.513,E2 26050.513} C_VEL
LIN {X 0,Y 703.129,Z 414.004,A -85,B 0,C 180,E1 26050.027,E2 26050.027} C_VEL
LIN {X 0,Y 701.027,Z 659.461,A -85,B 0,C 180,E1 26047.017,E2 26047.017} C_VEL
LIN {X 0,Y 699.573,Z 830.259,A -85,B 0,C 180,E1 26044.955,E2 26044.955} C_VEL
LIN {X 0,Y 699.073,Z 856.119,A -85,B 0,C 180,E1 26044.511,E2 26044.511} C_VEL
LIN {X 0,Y 698.354,Z 880.534,A -85,B 0,C 180,E1 26043.932,E2 26043.932} C_VEL
LIN {X 0,Y 697.647,Z 902.287,A -85,B 0,C 180,E1 26043.293,E2 26043.293} C_VEL
LIN {X 0,Y 696.747,Z 928.231,A -85,B 0,C 180,E1 26042.363,E2 26042.363} C_VEL
LIN {X 0,Y 695.86,Z 949.81,A -85,B 0,C 180,E1 26041.439,E2 26041.439} C_VEL
LIN {X 0,Y 695.016,Z 969.305,A -85,B 0,C 180,E1 26040.485,E2 26040.485} C_VEL
LIN {X 0,Y 693.947,Z 992.779,A -85,B 0,C 180,E1 26039.17,E2 26039.17} C_VEL
LIN {X 0,Y 693.034,Z 1012.943,A -85,B 0,C 180,E1 26037.869,E2 26037.869} C_VEL
LIN {X 0,Y 692.109,Z 1033.243,A -85,B 0,C 180,E1 26036.399,E2 26036.399} C_VEL
LIN {X 0,Y 691.236,Z 1052.547,A -85,B 0,C 180,E1 26034.802,E2 26034.802} C_VEL
LIN {X 0,Y 690.558,Z 1068.99,A -85,B 0,C 180,E1 26033.284,E2 26033.284} C_VEL
LIN {X 0,Y 689.821,Z 1087.65,A -85,B 0,C 180,E1 26031.335,E2 26031.335} C_VEL
LIN {X 0,Y 689.306,Z 1101.759,A -85,B 0,C 180,E1 26029.666,E2 26029.666} C_VEL
LIN {X 0,Y 688.844,Z 1116.739,A -85,B 0,C 180,E1 26027.66,E2 26027.66} C_VEL
LIN {X 0,Y 688.517,Z 1129.013,A -85,B 0,C 180,E1 26025.758,E2 26025.758} C_VEL
LIN {X 0,Y 688.278,Z 1139.213,A -85,B 0,C 180,E1 26023.955,E2 26023.955} C_VEL
LIN {X 0,Y 688.106,Z 1149.836,A -85,B 0,C 180,E1 26021.738,E2 26021.738} C_VEL
LIN {X 0,Y 687.992,Z 1156.91,A -85,B 0,C 180,E1 26019.959,E2 26019.959} C_VEL
LIN {X 0,Y 687.961,Z 1162.512,A -85,B 0,C 180,E1 26018.273,E2 26018.273} C_VEL
LIN {X 0,Y 687.932,Z 1167.456,A -85,B 0,C 180,E1 26016.426,E2 26016.426} C_VEL
LIN {X 0,Y 687.914,Z 1171.776,A -85,B 0,C 180,E1 26014.168,E2 26014.168} C_VEL
LIN {X 0,Y 687.914,Z 1173.901,A -85,B 0,C 180,E1 26012.333,E2 26012.333} C_VEL
LIN {X 0,Y 687.891,Z 1174.837,A -85,B 0,C 180,E1 26010.583,E2 26010.583} C_VEL
LIN {X 0,Y 687.911,Z 1174.637,A -85,B 0,C 180,E1 26008.584,E2 26008.584} C_VEL
LIN {X 0,Y 687.894,Z 1172.689,A -85,B 0,C 180,E1 26006.417,E2 26006.417} C_VEL
LIN {X 0,Y 687.915,Z 1169.905,A -85,B 0,C 180,E1 26004.659,E2 26004.659} C_VEL
LIN {X 0,Y 687.93,Z 1166.025,A -85,B 0,C 180,E1 26002.904,E2 26002.904} C_VEL
LIN {X 0,Y 687.99,Z 1159.968,A -85,B 0,C 180,E1 26000.801,E2 26000.801} C_VEL
LIN {X 0,Y 688.053,Z 1152.352,A -85,B 0,C 180,E1 25998.771,E2 25998.771} C_VEL
LIN {X 0,Y 688.188,Z 1144.784,A -85,B 0,C 180,E1 25997.071,E2 25997.071} C_VEL
LIN {X 0,Y 688.38,Z 1135.067,A -85,B 0,C 180,E1 25995.189,E2 25995.189} C_VEL
LIN {X 0,Y 688.697,Z 1121.983,A -85,B 0,C 180,E1 25993.033,E2 25993.033} C_VEL
LIN {X 0,Y 689.038,Z 1109.834,A -85,B 0,C 180,E1 25991.295,E2 25991.295} C_VEL
LIN {X 0,Y 689.552,Z 1094.63,A -85,B 0,C 180,E1 25989.369,E2 25989.369} C_VEL
LIN {X 0,Y 690.179,Z 1078.263,A -85,B 0,C 180,E1 25987.563,E2 25987.563} C_VEL
LIN {X 0,Y 690.911,Z 1060.622,A -85,B 0,C 180,E1 25985.823,E2 25985.823} C_VEL
LIN {X 0,Y 691.733,Z 1041.372,A -85,B 0,C 180,E1 25984.164,E2 25984.164} C_VEL
LIN {X 0,Y 692.58,Z 1022.624,A -85,B 0,C 180,E1 25982.718,E2 25982.718} C_VEL
LIN {X 0,Y 693.611,Z 1000.449,A -85,B 0,C 180,E1 25981.218,E2 25981.218} C_VEL
LIN {X 0,Y 694.477,Z 981.444,A -85,B 0,C 180,E1 25980.083,E2 25980.083} C_VEL
LIN {X 0,Y 695.491,Z 958.642,A -85,B 0,C 180,E1 25978.88,E2 25978.88} C_VEL
LIN {X 0,Y 696.468,Z 934.859,A -85,B 0,C 180,E1 25977.817,E2 25977.817} C_VEL
LIN {X 0,Y 697.265,Z 914.239,A -85,B 0,C 180,E1 25977.025,E2 25977.025} C_VEL
LIN {X 0,Y 698.147,Z 888.984,A -85,B 0,C 180,E1 25976.208,E2 25976.208} C_VEL
LIN {X 0,Y 698.779,Z 864.712,A -85,B 0,C 180,E1 25975.587,E2 25975.587} C_VEL
LIN {X 0,Y 699.312,Z 842.416,A -85,B 0,C 180,E1 25975.143,E2 25975.143} C_VEL
LIN {X 0,Y 699.802,Z 810.765,A -85,B 0,C 180,E1 25974.702,E2 25974.702} C_VEL
LIN {X 0,Y 701.749,Z 571.925,A -85,B 0,C 180,E1 25971.83,E2 25971.83} C_VEL
LIN {X 0,Y 703.03,Z 412.734,A -85,B 0,C 180,E1 25969.86,E2 25969.86} C_VEL
LIN {X 0,Y 699.322,Z 396.244,A -85,B 0,C 180,E1 25969.363,E2 25969.363} C_VEL
LIN {X 0,Y 700.849,Z 352.49,A -85,B 0,C 180,E1 25966.494,E2 25966.494} C_VEL
LIN {X 0,Y 701.074,Z 346.322,A -85,B 0,C 180,E1 25966.075,E2 25966.075} C_VEL
LIN {X 0,Y 693.921,Z 330.586,A -85,B 0,C 180,E1 25964.335,E2 25964.335} C_VEL
LIN {X 0,Y 690.05,Z 322.401,A -85,B 0,C 180,E1 25963.38,E2 25963.38} C_VEL
LIN {X 0,Y 688.446,Z 318.807,A -85,B 0,C 180,E1 25962.935,E2 25962.935} C_VEL
LIN {X 0,Y 688.466,Z 318.458,A -85,B 0,C 180,E1 25961.962,E2 25961.962} C_VEL
LIN {X 0,Y 688.409,Z 318.479,A -85,B 0,C 180,E1 25959.008,E2 25959.008} C_VEL
LIN {X 0,Y 688.437,Z 318.466,A -85,B 0,C 180,E1 25956.237,E2 25956.237} C_VEL
LIN {X 0,Y 688.427,Z 318.456,A -85,B 0,C 180,E1 25953.101,E2 25953.101} C_VEL
LIN {X 0,Y 688.432,Z 318.475,A -85,B 0,C 180,E1 25950.264,E2 25950.264} C_VEL
LIN {X 0,Y 688.453,Z 318.469,A -85,B 0,C 180,E1 25947.132,E2 25947.132} C_VEL
LIN {X 0,Y 688.436,Z 318.458,A -85,B 0,C 180,E1 25944.179,E2 25944.179} C_VEL
LIN {X 0,Y 688.465,Z 318.468,A -85,B 0,C 180,E1 25941.111,E2 25941.111} C_VEL
LIN {X 0,Y 688.44,Z 318.453,A -85,B 0,C 180,E1 25938.108,E2 25938.108} C_VEL
LIN {X 0,Y 688.461,Z 318.467,A -85,B 0,C 180,E1 25935.028,E2 25935.028} C_VEL
LIN {X 0,Y 688.447,Z 318.451,A -85,B 0,C 180,E1 25931.987,E2 25931.987} C_VEL
LIN {X 0,Y 688.454,Z 318.466,A -85,B 0,C 180,E1 25928.94,E2 25928.94} C_VEL
LIN {X 0,Y 688.449,Z 318.45,A -85,B 0,C 180,E1 25925.919,E2 25925.919} C_VEL
LIN {X 0,Y 688.443,Z 318.469,A -85,B 0,C 180,E1 25922.914,E2 25922.914} C_VEL
LIN {X 0,Y 688.451,Z 318.45,A -85,B 0,C 180,E1 25919.917,E2 25919.917} C_VEL
LIN {X 0,Y 688.432,Z 318.473,A -85,B 0,C 180,E1 25917.003,E2 25917.003} C_VEL
LIN {X 0,Y 688.455,Z 318.452,A -85,B 0,C 180,E1 25914.081,E2 25914.081} C_VEL
LIN {X 0,Y 688.431,Z 318.475,A -85,B 0,C 180,E1 25911.144,E2 25911.144} C_VEL
LIN {X 0,Y 688.459,Z 318.453,A -85,B 0,C 180,E1 25908.183,E2 25908.183} C_VEL
LIN {X 0,Y 688.43,Z 318.476,A -85,B 0,C 180,E1 25905.103,E2 25905.103} C_VEL
LIN {X 0,Y 688.435,Z 318.453,A -85,B 0,C 180,E1 25902.241,E2 25902.241} C_VEL
LIN {X 0,Y 688.428,Z 318.475,A -85,B 0,C 180,E1 25899.066,E2 25899.066} C_VEL
LIN {X 0,Y 688.413,Z 318.457,A -85,B 0,C 180,E1 25896.276,E2 25896.276} C_VEL
LIN {X 0,Y 688.452,Z 318.467,A -85,B 0,C 180,E1 25893.241,E2 25893.241} C_VEL
LIN {X 0,Y 688.395,Z 318.476,A -85,B 0,C 180,E1 25890.462,E2 25890.462} C_VEL
LIN {X 0,Y 688.447,Z 318.457,A -85,B 0,C 180,E1 25887.691,E2 25887.691} C_VEL
LIN {X 0,Y 688.395,Z 318.473,A -85,B 0,C 180,E1 25884.683,E2 25884.683} C_VEL
LIN {X 0,Y 688.384,Z 318.48,A -85,B 0,C 180,E1 25882.196,E2 25882.196} C_VEL
LIN {X 0,Y 688.454,Z 318.456,A -85,B 0,C 180,E1 25879.408,E2 25879.408} C_VEL
LIN {X 0,Y 688.435,Z 318.81,A -85,B 0,C 180,E1 25878.582,E2 25878.582} C_VEL
LIN {X 0,Y 689.817,Z 322.152,A -85,B 0,C 180,E1 25878.181,E2 25878.181} C_VEL
LIN {X 0,Y 693.441,Z 329.332,A -85,B 0,C 180,E1 25877.335,E2 25877.335} C_VEL
LIN {X 0,Y 701.168,Z 345.299,A -85,B 0,C 180,E1 25875.558,E2 25875.558} C_VEL
LIN {X 0,Y 702.279,Z 348.164,A -85,B 0,C 180,E1 25875.272,E2 25875.272} C_VEL
LIN {X 0,Y 702.44,Z 351.199,A -85,B 0,C 180,E1 25875.11,E2 25875.11} C_VEL
LIN {X 0,Y 706.575,Z 369.43,A -85,B 0,C 180,E1 25874.519,E2 25874.519} C_VEL
LIN {X 0,Y 704.445,Z 581.731,A -85,B 0,C 180,E1 25871.779,E2 25871.779} C_VEL
LIN {X 0,Y 702.366,Z 806.11,A -85,B 0,C 180,E1 25868.977,E2 25868.977} C_VEL
LIN {X 0,Y 701.861,Z 838.44,A -85,B 0,C 180,E1 25868.526,E2 25868.526} C_VEL
LIN {X 0,Y 701.17,Z 864.25,A -85,B 0,C 180,E1 25868.009,E2 25868.009} C_VEL
LIN {X 0,Y 700.396,Z 889.39,A -85,B 0,C 180,E1 25867.359,E2 25867.359} C_VEL
LIN {X 0,Y 699.347,Z 917.466,A -85,B 0,C 180,E1 25866.445,E2 25866.445} C_VEL
LIN {X 0,Y 698.407,Z 939.442,A -85,B 0,C 180,E1 25865.591,E2 25865.591} C_VEL
LIN {X 0,Y 697.473,Z 959.711,A -85,B 0,C 180,E1 25864.689,E2 25864.689} C_VEL
LIN {X 0,Y 696.516,Z 979.432,A -85,B 0,C 180,E1 25863.699,E2 25863.699} C_VEL
LIN {X 0,Y 695.399,Z 1001.888,A -85,B 0,C 180,E1 25862.432,E2 25862.432} C_VEL
LIN {X 0,Y 694.216,Z 1024.916,A -85,B 0,C 180,E1 25860.943,E2 25860.943} C_VEL
LIN {X 0,Y 693.267,Z 1043.783,A -85,B 0,C 180,E1 25859.576,E2 25859.576} C_VEL
LIN {X 0,Y 692.351,Z 1062.377,A -85,B 0,C 180,E1 25858.086,E2 25858.086} C_VEL
LIN {X 0,Y 691.305,Z 1083.589,A -85,B 0,C 180,E1 25856.176,E2 25856.176} C_VEL
LIN {X 0,Y 690.611,Z 1099.691,A -85,B 0,C 180,E1 25854.552,E2 25854.552} C_VEL
LIN {X 0,Y 689.908,Z 1116.492,A -85,B 0,C 180,E1 25852.675,E2 25852.675} C_VEL
LIN {X 0,Y 689.313,Z 1132.524,A -85,B 0,C 180,E1 25850.639,E2 25850.639} C_VEL
LIN {X 0,Y 688.907,Z 1145.026,A -85,B 0,C 180,E1 25848.857,E2 25848.857} C_VEL
LIN {X 0,Y 688.592,Z 1156.315,A -85,B 0,C 180,E1 25847.056,E2 25847.056} C_VEL
LIN {X 0,Y 688.307,Z 1168.607,A -85,B 0,C 180,E1 25844.813,E2 25844.813} C_VEL
LIN {X 0,Y 688.131,Z 1178.079,A -85,B 0,C 180,E1 25842.759,E2 25842.759} C_VEL
LIN {X 0,Y 688.006,Z 1186.016,A -85,B 0,C 180,E1 25840.751,E2 25840.751} C_VEL
LIN {X 0,Y 687.959,Z 1193.11,A -85,B 0,C 180,E1 25838.525,E2 25838.525} C_VEL
LIN {X 0,Y 687.926,Z 1198.594,A -85,B 0,C 180,E1 25836.258,E2 25836.258} C_VEL
LIN {X 0,Y 687.915,Z 1202.263,A -85,B 0,C 180,E1 25834.084,E2 25834.084} C_VEL
LIN {X 0,Y 687.907,Z 1204.438,A -85,B 0,C 180,E1 25831.832,E2 25831.832} C_VEL
LIN {X 0,Y 687.891,Z 1204.894,A -85,B 0,C 180,E1 25829.583,E2 25829.583} C_VEL
LIN {X 0,Y 687.907,Z 1203.958,A -85,B 0,C 180,E1 25827.501,E2 25827.501} C_VEL
LIN {X 0,Y 687.91,Z 1201.427,A -85,B 0,C 180,E1 25825.331,E2 25825.331} C_VEL
LIN {X 0,Y 687.927,Z 1197.151,A -85,B 0,C 180,E1 25823.071,E2 25823.071} C_VEL
LIN {X 0,Y 687.966,Z 1191.387,A -85,B 0,C 180,E1 25820.885,E2 25820.885} C_VEL
LIN {X 0,Y 688.04,Z 1184.276,A -85,B 0,C 180,E1 25818.771,E2 25818.771} C_VEL
LIN {X 0,Y 688.2,Z 1173.937,A -85,B 0,C 180,E1 25816.301,E2 25816.301} C_VEL
LIN {X 0,Y 688.395,Z 1164.292,A -85,B 0,C 180,E1 25814.368,E2 25814.368} C_VEL
LIN {X 0,Y 688.644,Z 1154.224,A -85,B 0,C 180,E1 25812.596,E2 25812.596} C_VEL
LIN {X 0,Y 688.984,Z 1142.515,A -85,B 0,C 180,E1 25810.766,E2 25810.766} C_VEL
LIN {X 0,Y 689.531,Z 1126.509,A -85,B 0,C 180,E1 25808.566,E2 25808.566} C_VEL
LIN {X 0,Y 690.12,Z 1111.233,A -85,B 0,C 180,E1 25806.72,E2 25806.72} C_VEL
LIN {X 0,Y 690.812,Z 1094.566,A -85,B 0,C 180,E1 25804.907,E2 25804.907} C_VEL
LIN {X 0,Y 691.749,Z 1074.828,A -85,B 0,C 180,E1 25803.008,E2 25803.008} C_VEL
LIN {X 0,Y 692.544,Z 1057.943,A -85,B 0,C 180,E1 25801.546,E2 25801.546} C_VEL
LIN {X 0,Y 693.498,Z 1038.97,A -85,B 0,C 180,E1 25800.058,E2 25800.058} C_VEL
LIN {X 0,Y 694.72,Z 1015.164,A -85,B 0,C 180,E1 25798.406,E2 25798.406} C_VEL
LIN {X 0,Y 695.722,Z 995.431,A -85,B 0,C 180,E1 25797.192,E2 25797.192} C_VEL
LIN {X 0,Y 696.698,Z 975.859,A -85,B 0,C 180,E1 25796.113,E2 25796.113} C_VEL
LIN {X 0,Y 697.765,Z 953.688,A -85,B 0,C 180,E1 25795.027,E2 25795.027} C_VEL
LIN {X 0,Y 698.899,Z 927.081,A -85,B 0,C 180,E1 25793.911,E2 25793.911} C_VEL
LIN {X 0,Y 699.792,Z 904.845,A -85,B 0,C 180,E1 25793.122,E2 25793.122} C_VEL
LIN {X 0,Y 700.635,Z 881.918,A -85,B 0,C 180,E1 25792.433,E2 25792.433} C_VEL
LIN {X 0,Y 701.467,Z 854.937,A -85,B 0,C 180,E1 25791.784,E2 25791.784} C_VEL
LIN {X 0,Y 702.07,Z 827.582,A -85,B 0,C 180,E1 25791.303,E2 25791.303} C_VEL
LIN {X 0,Y 704.214,Z 605.362,A -85,B 0,C 180,E1 25788.52,E2 25788.52} C_VEL
LIN {X 0,Y 706.224,Z 401.968,A -85,B 0,C 180,E1 25785.906,E2 25785.906} C_VEL
LIN {X 0,Y 706.438,Z 368.104,A -85,B 0,C 180,E1 25785.451,E2 25785.451} C_VEL
LIN {X 0,Y 702.256,Z 350.015,A -85,B 0,C 180,E1 25784.842,E2 25784.842} C_VEL
LIN {X 0,Y 702.115,Z 347.242,A -85,B 0,C 180,E1 25784.652,E2 25784.652} C_VEL
LIN {X 0,Y 693.807,Z 330.063,A -85,B 0,C 180,E1 25782.749,E2 25782.749} C_VEL
LIN {X 0,Y 689.816,Z 322.153,A -85,B 0,C 180,E1 25781.819,E2 25781.819} C_VEL
LIN {X 0,Y 688.42,Z 318.723,A -85,B 0,C 180,E1 25781.399,E2 25781.399} C_VEL
LIN {X 0,Y 688.41,Z 318.467,A -85,B 0,C 180,E1 25779.14,E2 25779.14} C_VEL
LIN {X 0,Y 688.397,Z 318.465,A -85,B 0,C 180,E1 25775.999,E2 25775.999} C_VEL
LIN {X 0,Y 688.39,Z 318.471,A -85,B 0,C 180,E1 25773.401,E2 25773.401} C_VEL
LIN {X 0,Y 688.47,Z 318.474,A -85,B 0,C 180,E1 25770.455,E2 25770.455} C_VEL
LIN {X 0,Y 688.397,Z 318.462,A -85,B 0,C 180,E1 25767.603,E2 25767.603} C_VEL
LIN {X 0,Y 688.429,Z 318.476,A -85,B 0,C 180,E1 25764.911,E2 25764.911} C_VEL
LIN {X 0,Y 688.421,Z 318.47,A -85,B 0,C 180,E1 25761.739,E2 25761.739} C_VEL
LIN {X 0,Y 688.419,Z 318.469,A -85,B 0,C 180,E1 25758.987,E2 25758.987} C_VEL
LIN {X 0,Y 688.461,Z 318.469,A -85,B 0,C 180,E1 25755.932,E2 25755.932} C_VEL
LIN {X 0,Y 688.416,Z 318.468,A -85,B 0,C 180,E1 25753.096,E2 25753.096} C_VEL
LIN {X 0,Y 688.46,Z 318.473,A -85,B 0,C 180,E1 25750.206,E2 25750.206} C_VEL
LIN {X 0,Y 688.426,Z 318.463,A -85,B 0,C 180,E1 25747.253,E2 25747.253} C_VEL
LIN {X 0,Y 688.46,Z 318.466,A -85,B 0,C 180,E1 25744.331,E2 25744.331} C_VEL
LIN {X 0,Y 688.44,Z 318.463,A -85,B 0,C 180,E1 25741.248,E2 25741.248} C_VEL
LIN {X 0,Y 688.46,Z 318.463,A -85,B 0,C 180,E1 25738.252,E2 25738.252} C_VEL
LIN {X 0,Y 688.45,Z 318.463,A -85,B 0,C 180,E1 25735.168,E2 25735.168} C_VEL
LIN {X 0,Y 688.458,Z 318.462,A -85,B 0,C 180,E1 25732.096,E2 25732.096} C_VEL
LIN {X 0,Y 688.455,Z 318.463,A -85,B 0,C 180,E1 25729.032,E2 25729.032} C_VEL
LIN {X 0,Y 688.451,Z 318.466,A -85,B 0,C 180,E1 25725.963,E2 25725.963} C_VEL
LIN {X 0,Y 688.46,Z 318.463,A -85,B 0,C 180,E1 25722.94,E2 25722.94} C_VEL
LIN {X 0,Y 688.446,Z 318.472,A -85,B 0,C 180,E1 25719.866,E2 25719.866} C_VEL
LIN {X 0,Y 688.462,Z 318.459,A -85,B 0,C 180,E1 25716.822,E2 25716.822} C_VEL
LIN {X 0,Y 688.438,Z 318.477,A -85,B 0,C 180,E1 25713.705,E2 25713.705} C_VEL
LIN {X 0,Y 688.459,Z 318.468,A -85,B 0,C 180,E1 25712.364,E2 25712.364} C_VEL
LIN {X 0,Y 687.461,Z 318.581,A -85,B 0,C 180,E1 25711.723,E2 25711.723} C_VEL
LIN {X 0,Y 681.028,Z 319.398,A -85,B 0,C 180,E1 25709.927,E2 25709.927} C_VEL
LIN {X 0,Y 680.486,Z 319.466,A -85,B 0,C 180,E1 25709.46,E2 25709.46} C_VEL
LIN {X 0,Y 680.52,Z 319.438,A -85,B 0,C 180,E1 25706.565,E2 25706.565} C_VEL
LIN {X 0,Y 680.483,Z 319.452,A -85,B 0,C 180,E1 25703.48,E2 25703.48} C_VEL
LIN {X 0,Y 680.502,Z 319.466,A -85,B 0,C 180,E1 25700.598,E2 25700.598} C_VEL
LIN {X 0,Y 680.534,Z 319.684,A -85,B 0,C 180,E1 25697.659,E2 25697.659} C_VEL
LIN {X 0,Y 681.83,Z 323.037,A -85,B 0,C 180,E1 25697.236,E2 25697.236} C_VEL
LIN {X 0,Y 686.762,Z 333.129,A -85,B 0,C 180,E1 25696.013,E2 25696.013} C_VEL
LIN {X 0,Y 693.845,Z 348.69,A -85,B 0,C 180,E1 25694.256,E2 25694.256} C_VEL
LIN {X 0,Y 694.632,Z 350.69,A -85,B 0,C 180,E1 25694.047,E2 25694.047} C_VEL
LIN {X 0,Y 692.845,Z 393.148,A -85,B 0,C 180,E1 25691.208,E2 25691.208} C_VEL
LIN {X 0,Y 692.915,Z 397.324,A -85,B 0,C 180,E1 25690.969,E2 25690.969} C_VEL
LIN {X 0,Y 696.982,Z 415.856,A -85,B 0,C 180,E1 25690.429,E2 25690.429} C_VEL
LIN {X 0,Y 694.629,Z 660.403,A -85,B 0,C 180,E1 25687.405,E2 25687.405} C_VEL
LIN {X 0,Y 693.008,Z 830.303,A -85,B 0,C 180,E1 25685.336,E2 25685.336} C_VEL
LIN {X 0,Y 692.446,Z 856.368,A -85,B 0,C 180,E1 25684.883,E2 25684.883} C_VEL
LIN {X 0,Y 691.671,Z 880.445,A -85,B 0,C 180,E1 25684.309,E2 25684.309} C_VEL
LIN {X 0,Y 690.905,Z 901.774,A -85,B 0,C 180,E1 25683.679,E2 25683.679} C_VEL
LIN {X 0,Y 689.907,Z 927.111,A -85,B 0,C 180,E1 25682.773,E2 25682.773} C_VEL
LIN {X 0,Y 688.921,Z 948.814,A -85,B 0,C 180,E1 25681.842,E2 25681.842} C_VEL
LIN {X 0,Y 687.969,Z 968.668,A -85,B 0,C 180,E1 25680.867,E2 25680.867} C_VEL
LIN {X 0,Y 686.801,Z 991.718,A -85,B 0,C 180,E1 25679.573,E2 25679.573} C_VEL
LIN {X 0,Y 685.701,Z 1012.952,A -85,B 0,C 180,E1 25678.194,E2 25678.194} C_VEL
LIN {X 0,Y 684.69,Z 1032.964,A -85,B 0,C 180,E1 25676.73,E2 25676.73} C_VEL
LIN {X 0,Y 683.679,Z 1052.553,A -85,B 0,C 180,E1 25675.095,E2 25675.095} C_VEL
LIN {X 0,Y 682.918,Z 1068.994,A -85,B 0,C 180,E1 25673.56,E2 25673.56} C_VEL
LIN {X 0,Y 682.076,Z 1087.657,A -85,B 0,C 180,E1 25671.589,E2 25671.589} C_VEL
LIN {X 0,Y 681.497,Z 1102.018,A -85,B 0,C 180,E1 25669.868,E2 25669.868} C_VEL
LIN {X 0,Y 680.956,Z 1117.325,A -85,B 0,C 180,E1 25667.783,E2 25667.783} C_VEL
LIN {X 0,Y 680.602,Z 1129.018,A -85,B 0,C 180,E1 25665.946,E2 25665.946} C_VEL
LIN {X 0,Y 680.339,Z 1139.214,A -85,B 0,C 180,E1 25664.121,E2 25664.121} C_VEL
LIN {X 0,Y 680.131,Z 1149.839,A -85,B 0,C 180,E1 25661.878,E2 25661.878} C_VEL
LIN {X 0,Y 680.004,Z 1157.217,A -85,B 0,C 180,E1 25659.992,E2 25659.992} C_VEL
LIN {X 0,Y 679.965,Z 1163.024,A -85,B 0,C 180,E1 25658.201,E2 25658.201} C_VEL
LIN {X 0,Y 679.918,Z 1168.623,A -85,B 0,C 180,E1 25655.993,E2 25655.993} C_VEL
LIN {X 0,Y 679.916,Z 1172.117,A -85,B 0,C 180,E1 25653.963,E2 25653.963} C_VEL
LIN {X 0,Y 679.914,Z 1174.036,A -85,B 0,C 180,E1 25652.191,E2 25652.191} C_VEL
LIN {X 0,Y 679.897,Z 1174.926,A -85,B 0,C 180,E1 25650.253,E2 25650.253} C_VEL
LIN {X 0,Y 679.912,Z 1174.244,A -85,B 0,C 180,E1 25647.978,E2 25647.978} C_VEL
LIN {X 0,Y 679.91,Z 1172.35,A -85,B 0,C 180,E1 25646.121,E2 25646.121} C_VEL
LIN {X 0,Y 679.906,Z 1169.274,A -85,B 0,C 180,E1 25644.261,E2 25644.261} C_VEL
LIN {X 0,Y 679.961,Z 1164.057,A -85,B 0,C 180,E1 25642.055,E2 25642.055} C_VEL
LIN {X 0,Y 679.994,Z 1157.844,A -85,B 0,C 180,E1 25640.094,E2 25640.094} C_VEL
LIN {X 0,Y 680.116,Z 1150.926,A -85,B 0,C 180,E1 25638.295,E2 25638.295} C_VEL
LIN {X 0,Y 680.294,Z 1141.509,A -85,B 0,C 180,E1 25636.226,E2 25636.226} C_VEL
LIN {X 0,Y 680.576,Z 1130.077,A -85,B 0,C 180,E1 25634.142,E2 25634.142} C_VEL
LIN {X 0,Y 680.891,Z 1118.975,A -85,B 0,C 180,E1 25632.376,E2 25632.376} C_VEL
LIN {X 0,Y 681.421,Z 1103.873,A -85,B 0,C 180,E1 25630.276,E2 25630.276} C_VEL
LIN {X 0,Y 681.986,Z 1089.99,A -85,B 0,C 180,E1 25628.589,E2 25628.589} C_VEL
LIN {X 0,Y 682.699,Z 1073.53,A -85,B 0,C 180,E1 25626.798,E2 25626.798} C_VEL
LIN {X 0,Y 683.569,Z 1055.07,A -85,B 0,C 180,E1 25625.039,E2 25625.039} C_VEL
LIN {X 0,Y 684.408,Z 1037.976,A -85,B 0,C 180,E1 25623.582,E2 25623.582} C_VEL
LIN {X 0,Y 685.555,Z 1016.089,A -85,B 0,C 180,E1 25621.934,E2 25621.934} C_VEL
LIN {X 0,Y 686.529,Z 996.787,A -85,B 0,C 180,E1 25620.654,E2 25620.654} C_VEL
LIN {X 0,Y 687.715,Z 973.893,A -85,B 0,C 180,E1 25619.315,E2 25619.315} C_VEL
LIN {X 0,Y 688.791,Z 951.683,A -85,B 0,C 180,E1 25618.201,E2 25618.201} C_VEL
LIN {X 0,Y 689.713,Z 931.45,A -85,B 0,C 180,E1 25617.316,E2 25617.316} C_VEL
LIN {X 0,Y 690.736,Z 907.18,A -85,B 0,C 180,E1 25616.405,E2 25616.405} C_VEL
LIN {X 0,Y 691.581,Z 882.667,A -85,B 0,C 180,E1 25615.66,E2 25615.66} C_VEL
LIN {X 0,Y 692.284,Z 860.693,A -85,B 0,C 180,E1 25615.122,E2 25615.122} C_VEL
LIN {X 0,Y 692.966,Z 834.164,A -85,B 0,C 180,E1 25614.629,E2 25614.629} C_VEL
LIN {X 0,Y 693.482,Z 786.017,A -85,B 0,C 180,E1 25614.022,E2 25614.022} C_VEL
LIN {X 0,Y 695.577,Z 557.375,A -85,B 0,C 180,E1 25611.241,E2 25611.241} C_VEL
LIN {X 0,Y 696.883,Z 414.578,A -85,B 0,C 180,E1 25609.457,E2 25609.457} C_VEL
LIN {X 0,Y 692.766,Z 396.085,A -85,B 0,C 180,E1 25608.888,E2 25608.888} C_VEL
LIN {X 0,Y 694.515,Z 353.321,A -85,B 0,C 180,E1 25606.042,E2 25606.042} C_VEL
LIN {X 0,Y 694.483,Z 350.098,A -85,B 0,C 180,E1 25605.808,E2 25605.808} C_VEL
LIN {X 0,Y 687.725,Z 335.246,A -85,B 0,C 180,E1 25604.141,E2 25604.141} C_VEL
LIN {X 0,Y 683.601,Z 326.744,A -85,B 0,C 180,E1 25603.125,E2 25603.125} C_VEL
LIN {X 0,Y 681.744,Z 322.913,A -85,B 0,C 180,E1 25602.657,E2 25602.657} C_VEL
LIN {X 0,Y 680.53,Z 319.633,A -85,B 0,C 180,E1 25602.226,E2 25602.226} C_VEL
LIN {X 0,Y 680.48,Z 319.468,A -85,B 0,C 180,E1 25599.186,E2 25599.186} C_VEL
LIN {X 0,Y 680.485,Z 319.453,A -85,B 0,C 180,E1 25596.37,E2 25596.37} C_VEL
LIN {X 0,Y 680.502,Z 319.44,A -85,B 0,C 180,E1 25593.235,E2 25593.235} C_VEL
LIN {X 0,Y 680.488,Z 319.466,A -85,B 0,C 180,E1 25590.362,E2 25590.362} C_VEL
LIN {X 0,Y 680.524,Z 319.458,A -85,B 0,C 180,E1 25587.264,E2 25587.264} C_VEL
LIN {X 0,Y 680.49,Z 319.447,A -85,B 0,C 180,E1 25584.294,E2 25584.294} C_VEL
LIN {X 0,Y 680.522,Z 319.459,A -85,B 0,C 180,E1 25581.28,E2 25581.28} C_VEL
LIN {X 0,Y 680.491,Z 319.44,A -85,B 0,C 180,E1 25578.327,E2 25578.327} C_VEL
LIN {X 0,Y 680.513,Z 319.462,A -85,B 0,C 180,E1 25575.423,E2 25575.423} C_VEL
LIN {X 0,Y 680.5,Z 319.435,A -85,B 0,C 180,E1 25572.474,E2 25572.474} C_VEL
LIN {X 0,Y 680.513,Z 319.462,A -85,B 0,C 180,E1 25569.472,E2 25569.472} C_VEL
LIN {X 0,Y 680.513,Z 319.433,A -85,B 0,C 180,E1 25566.496,E2 25566.496} C_VEL
LIN {X 0,Y 680.512,Z 319.464,A -85,B 0,C 180,E1 25563.454,E2 25563.454} C_VEL
